rr := RDM(rr);
(* generate random date and randon dt *)
xdt := DWORD_TO_DT(rx);

(* analyze date *)
s1 := DT_TO_STRING(xdt);
s1 := RIGHT(s1, LEN(s1)-FIND(s1,'#'));
yr := STRING_TO_INT(LEFT(s1,4));
s1 := RIGHT(s1, LEN(s1)-FIND(s1,'-'));
mth := STRING_TO_INT(LEFT(s1,2));
s1 := RIGHT(s1, LEN(s1)-FIND(s1,'-'));
day := STRING_TO_INT(LEFT(s1,2));
(* analyze Time *)
s1 := RIGHT(s1, LEN(s1)-FIND(s1,'-'));
hr := STRING_TO_INT(LEFT(s1,2));
s1 := RIGHT(s1, LEN(s1)-FIND(s1,':'));
m := STRING_TO_INT(LEFT(s1,2));
s1 := RIGHT(s1, LEN(s1)-FIND(s1,':'));
sec := STRING_TO_INT(LEFT(s1,2));

(*
xd := DT_TO_DATE(xdt);
dt_to Date delivers wrong result when year > 2038
*)
xd := set_Date(yr,mth,day);

(* test set_date *)
test := 'set_date';
IF set_Date(yr,mth,day) <> xd THEN RETURN; END_IF;

(* test set_dt *)
test := 'set_dt';
IF set_DT(yr,mth,day,hr,m,sec) <> xdt THEN RETURN; END_IF;

(* test date_add *)
test := 'date_add';
YD := date_add(xd,0,0,0,0);
IF YD <> XD THEN RETURN; END_IF;
yd := date_add(d#2000-1-1,5,0,0,0);
IF yd <> d#2000-1-6 THEN RETURN; END_IF;
yd := date_add(d#2000-1-1,-31,0,0,0);
IF yd <> d#1999-12-1 THEN RETURN; END_IF;
yd := date_add(d#2000-1-1,60,0,0,0);
IF yd <> d#2000-3-1 THEN RETURN; END_IF;
yd := date_add(d#2001-1-1,59,0,0,0);
IF yd <> d#2001-3-1 THEN RETURN; END_IF;
yd := date_add(d#2002-1-1,59,0,0,0);
IF yd <> d#2002-3-1 THEN RETURN; END_IF;
yd := date_add(d#2003-1-1,59,0,0,0);
IF yd <> d#2003-3-1 THEN RETURN; END_IF;
yd := date_add(d#2004-1-1,60,0,0,0);
IF yd <> d#2004-3-1 THEN RETURN; END_IF;
yd := date_add(d#2000-1-1,0,1,0,0);
IF yd <> d#2000-1-8 THEN RETURN; END_IF;
yd := date_add(d#2000-1-1,0,-1,0,0);
IF yd <> d#1999-12-25 THEN RETURN; END_IF;
yd := date_add(d#2000-1-1,0,0,12,0);
IF yd <> d#2001-1-1 THEN RETURN; END_IF;
yd := date_add(d#2000-1-1,0,0,-1,0);
IF yd <> d#1999-12-1 THEN RETURN; END_IF;
yd := date_add(d#2000-1-1,0,0,0,99);
IF yd <> d#2099-1-1 THEN RETURN; END_IF;
yd := date_add(d#2000-1-1,0,0,0,-12);
IF yd <> d#1988-1-1 THEN RETURN; END_IF;
yd := date_add(d#2000-1-1,-31,1,1,1);
IF yd <> d#2001-1-8 THEN RETURN; END_IF;
yd := date_add(d#2000-1-1,31,1,-1,-1);
IF yd <> d#1999-1-8 THEN RETURN; END_IF;

(* test day_of_date *)
test := 'day_of_date';
IF day_of_date(XD) <> DATE_TO_DWORD(xd) / 86400 THEN RETURN; END_IF;

(* test day_of_month *)
test := 'day_of_month';
IF day_of_month(xd) <> day THEN RETURN; END_IF;

(* test day_of_year *)
test := 'day_of_year';
IF day_of_date(xd) - day_of_date(set_Date(yr,1,1)) + 1 <> day_of_year(xd) THEN RETURN; END_IF;

(* test days_delta *)
test := 'days_delta';
IF days_delta(xd, xd) <> 0 THEN RETURN; END_IF;
IF days_delta(D#2008-1-1,D#2007-12-31) <> -1 THEN RETURN; END_IF;
IF days_delta(D#2008-2-28,D#2008-3-1) <> 2 THEN RETURN; END_IF;
IF days_delta(D#2012-3-1,D#2012-2-28) <> -2 THEN RETURN; END_IF;
IF days_delta(D#2007-2-28,D#2007-3-1) <> 1 THEN RETURN; END_IF;
IF days_delta(D#1970-1-1,xd) <> day_of_date(xd) THEN RETURN; END_IF;

(* test DST *)
(*
Equation used TO calculate the beginning OF European Summer TIME:
Sunday (31 - (5*y/4 + 4) mod 7) March at 01.00 UTC
(valid through 2099, courtesy of Robert H. van Gent, EC).
European Summer Time ends (clocks go back) at 01.00 UTC on

    * 29 October 2006
    * 28 October 2007
    * 26 October 2008

Equation used to calculate the end of European Summer Time:
Sunday (31 - (5*y/4 + 1) mod 7) October at 01.00 UTC
(validity AND credits as above).
*)
test := 'dst';
ti := 31 -(5*yr/4 + 4) MOD 7;
te := 31-(5*yr/4+1) MOD 7;
tdt := set_DT(yr,3,ti,1,0,0);
tde := set_DT(yr,10,te,1,0,0);
tb := xdt >= tdt AND xdt < tde;
IF DST(xdt) <> tb THEN RETURN; END_IF;
IF DST(tdt) = FALSE THEN RETURN; END_IF;
tdt := set_DT(yr,3,ti,0,59,59);
IF DST(tdt) = TRUE THEN RETURN; END_IF;
tdt := set_DT(yr,10,te,0,59,59);
IF DST(tdt) = FALSE THEN RETURN; END_IF;
IF DST(tde) = TRUE THEN RETURN; END_IF;

(* easter test *)
test := 'easter';
IF easter_test() <> TRUE THEN RETURN; END_IF;

(* test leap_of_date *)
test := 'leap_of_Date';
tb := yr MOD 4 = 0;
IF leap_of_Date(xd) <> tb THEN RETURN; END_IF;

(* test leap_year *)
test := 'leap_year';
IF leap_year(yr) <> tb THEN RETURN; END_IF;

(* test local_time *)
test := 'local_time';
TT := T#12h;
IF local_time(xdt,-12,FALSE) <> xdt - TT THEN RETURN; END_IF;
IF local_time(xdt,0,FALSE) <> xdt THEN RETURN; END_IF;
TT := T#1h;
IF local_time(xdt,1,FALSE) <> xdt + TT THEN RETURN; END_IF;
TT := T#12h;
IF local_time(xdt,+12,FALSE) <> xdt + TT THEN RETURN; END_IF;
IF DST(xdt) THEN
	TT := T#11h;
	IF local_time(xdt,-12,TRUE) <> xdt - TT THEN RETURN; END_IF;
	TT := T#1h;
	IF local_time(xdt,0,TRUE) <> xdt + TT THEN RETURN; END_IF;
	TT := T#2h;
	IF local_time(xdt,1,TRUE) <> xdt + TT THEN RETURN; END_IF;
	TT := T#13h;
	IF local_time(xdt,+12,TRUE) <> xdt + TT THEN RETURN; END_IF;
ELSE
	TT := T#12h;
	IF local_time(xdt,-12,TRUE) <> xdt - TT THEN RETURN; END_IF;
	IF local_time(xdt,0,TRUE) <> xdt THEN RETURN; END_IF;
	TT := T#1h;
	IF local_time(xdt,1,TRUE) <> xdt + TT THEN RETURN; END_IF;
	TT := T#12h;
	IF local_time(xdt,+12,TRUE) <> xdt + TT THEN RETURN; END_IF;
END_IF;

(* ltime_to_utc *)
test := 'ltime_to_utc';
TT := T#1h;
IF Ltime_to_UTC(xdt+TT,FALSE,1) <> xdt THEN RETURN; END_IF;
IF Ltime_to_UTC(xdt - TT, FALSE,-1) <> xdt THEN RETURN; END_IF;
IF Ltime_to_UTC(xdt, FALSE,0) <> xdt THEN RETURN; END_IF;
TT := T#2h;
IF Ltime_to_UTC(xdt+ TT,TRUE,1) <> xdt THEN RETURN; END_IF;
IF Ltime_to_UTC(xdt, TRUE,-1) <> xdt THEN RETURN; END_IF;
TT := T#1h;
IF Ltime_to_UTC(xdt + TT, TRUE,0) <> xdt THEN RETURN; END_IF;

(* month test *)
test := 'month';
IF month(xd) <> mth THEN RETURN; END_IF;

(* period test *)
test := 'period';
yd := set_Date(2000,mth,day);
IF period(d#2000-3-3,xd,d#2000-9-3) <> (yd >= d#2000-3-3 AND yd <= d#2000-9-3) THEN RETURN; END_IF;
IF period(d#2000-9-3,xd,d#2000-3-3) <> (yd <= d#2000-3-3 OR yd >= d#2000-9-3) THEN RETURN; END_IF;

(* test weekday *)
test := 'weekday';
wd := weekday(xd);
wdi := DWORD_TO_DINT(DATE_TO_DWORD(xd)/86400);
wdi := (wdi + 4) MOD 7;
IF wdi = 0 THEN wdi := 7; END_IF;
IF wd <> wdi THEN RETURN; END_IF;

(* test year *)
test := 'year';
IF year(xd) <> yr THEN RETURN; END_IF;

(* test year_begin *)
test := 'year_begin';
IF year_begin(yr) <> set_Date(yr,1,1) THEN RETURN; END_IF;

(* test work_week *)
test := 'work_week';
IF NOT work_week_test() THEN RETURN; END_IF;

(* set output true if there are no errors *)
test := 'finished';
good := TRUE;


(* revision history
hm		26. mar. 2008		rev 1.0
	original release

*)
END_FUNCTION_BLOCK

(* POU Mathematical/RDMDW, ST *)
FUNCTION RDMDW : DWORD
VAR_INPUT
	last : DWORD;
END_VAR
VAR
	RX: REAL;
	M: REAL;
END_VAR




(*
version 1.0	14. mar 2008
programmer 	hugo
tested by		tobias

this function calculates a DWORD pseudo random number.

*)
M := BIT_COUNT(last);
RX := RDM(FRACT(M*pi1));
RDMDW := SHL(REAL_TO_DWORD(rx*65535),16);
RX := RDM(FRACT(M*e));
RDMDW := RDMDW OR (REAL_TO_DWORD(rx*65535) AND 16#0000FFFF);



(* revision history
hm		14. mar 2008		rev 1.0
	original version

*)
END_FUNCTION

(* POU Time&Date/set_Date, ST *)
FUNCTION set_Date : DATE
VAR_INPUT
	year : INT;
	month : INT;
	day : INT;
END_VAR
VAR
	count : DWORD;
END_VAR

(*
version 1.5	16. mar. 2008
programmer 	hugo
tested by		tobias

creates a date output from year, month and day of month   

*)
IF STEP7 THEN
	count := SHR(INT_TO_DWORD(year) * 1461 - 2907393,2)+INT_TO_DWORD(day);
ELSE
	count := SHR(INT_TO_DWORD(year) * 1461 - 2878173,2)+INT_TO_DWORD(day);
END_IF;

IF month < 5 THEN
	IF month < 3 THEN
		IF month = 2 THEN count := count + 31; END_IF;
	ELSE
		IF month = 4 THEN
			IF SHL(year,14) = 0 THEN count := count + 91; ELSE count := count + 90; END_IF;
		ELSE (* month = 3 *)
			IF SHL(year,14) = 0 THEN count := count + 60; ELSE count := count + 59; END_IF;
		END_IF;
	END_IF;
ELSIF month < 9 THEN
	IF month < 7 THEN
		IF month = 6 THEN
			IF SHL(year,14) = 0 THEN count := count + 152; ELSE count := count + 151; END_IF;
		ELSE (* month = 5 *)
			IF SHL(year,14) = 0 THEN count := count + 121; ELSE count := count + 120; END_IF;
		END_IF;
	ELSE
		IF month = 8 THEN
			IF SHL(year,14) = 0 THEN count := count + 213; ELSE count := count + 212; END_IF;
		ELSE (* month = 7 *)
			IF SHL(year,14) = 0 THEN count := count + 182; ELSE count := count + 181; END_IF;
		END_IF;
	END_IF;
ELSE (* month is 9 or higher *)
	IF month < 11 THEN
		IF month = 10 THEN
			IF SHL(year,14) = 0 THEN count := count + 274; ELSE count := count + 273; END_IF;
		ELSE (* month = 9 *)
			IF SHL(year,14) = 0 THEN count := count + 244; ELSE count := count + 243; END_IF;
		END_IF;
	ELSE
		IF month = 12 THEN
			IF SHL(year,14) = 0 THEN count := count + 335; ELSE count := count + 334; END_IF;
		ELSE (* month = 11 *)
			IF SHL(year,14) = 0 THEN count := count + 305; ELSE count := count + 304; END_IF;
		END_IF;
	END_IF;
END_IF;
set_Date := DWORD_TO_DATE(count * 86400);

(*  code before rev 1.4
leap := leap_year(year);
IF STEP7 THEN
	count := SHR((year-1)*1461-2905932+day*4,2);
ELSE
	count := SHR((year-1)*1461-2876712+day*4,2);
END_IF;
CASE month OF
2:	count := count + 31;
3:	IF leap THEN count := count + 60; ELSE count := count + 59; END_IF;
4:	IF leap THEN count := count + 91; ELSE count := count + 90; END_IF;
5:	IF leap THEN count := count + 121; ELSE count := count + 120; END_IF;
6:	IF leap THEN count := count + 152; ELSE count := count + 151; END_IF;
7:	IF leap THEN count := count + 182; ELSE count := count + 181; END_IF;
8:	IF leap THEN count := count + 213; ELSE count := count + 212; END_IF;
9:	IF leap THEN count := count + 244; ELSE count := count + 243; END_IF;
10:	IF leap THEN count := count + 274; ELSE count := count + 273; END_IF;
11:	IF leap THEN count := count + 305; ELSE count := count + 304; END_IF;
12:	IF leap THEN count := count + 335; ELSE count := count + 334; END_IF;
END_CASE;
set_Date := DWORD_TO_DATE(count * 86400);
*)

(* old code before rev 1.3
leap := leap_year(year);
IF STEP7 THEN
	count := TRUNC((year-1)*365.25-726483+day);
ELSE
	count := TRUNC((year-1)*365.25-719178+day);
END_IF;
CASE month OF
2:	count := count + 31;
3:	IF leap THEN count := count + 60; ELSE count := count + 59; END_IF;
4:	IF leap THEN count := count + 91; ELSE count := count + 90; END_IF;
5:	IF leap THEN count := count + 121; ELSE count := count + 120; END_IF;
6:	IF leap THEN count := count + 152; ELSE count := count + 151; END_IF;
7:	IF leap THEN count := count + 182; ELSE count := count + 181; END_IF;
8:	IF leap THEN count := count + 213; ELSE count := count + 212; END_IF;
9:	IF leap THEN count := count + 244; ELSE count := count + 243; END_IF;
10:	IF leap THEN count := count + 274; ELSE count := count + 273; END_IF;
11:	IF leap THEN count := count + 305; ELSE count := count + 304; END_IF;
12:	IF leap THEN count := count + 335; ELSE count := count + 334; END_IF;
END_CASE;
set_Date := DWORD_TO_DATE(count * 86400);
*)




(* revision history
hm	4. aug. 2006	rev 1.0
	original version

hm	19 sep. 2007	rev 1.1
	use function leap_year to calculate leap year, more exceptions are handled

hm	1. okt	2007	rev 1.2
	added compatibility to step7

hm	16.dec 2007	rev 1.3
	changed code to improove performance

hm	3. jan. 2008	rev 1.4
	further improvements in performance

hm	16. mar. 2008	rev 1.5
	added type conversions to avoid warnings under codesys 3.0
*)
END_FUNCTION

(* POU Time&Date/year, ST *)
FUNCTION year : INT
VAR_INPUT
	idate : DATE;
END_VAR
VAR
END_VAR

(*
version 1.2	23 dec 2007
programmer 	hugo
tested by		tobias

returs the year of a date  
the function works for dates from 1970 - 2099 

*)
IF Step7 THEN
	year := DWORD_TO_INT((DATE_TO_DWORD(idate)+43200) / 31557600 + 1990);
ELSE
	year := DWORD_TO_INT((DATE_TO_DWORD(idate)+43200) / 31557600 + 1970);
END_IF;

(* code used prior to rev 1.1
year := DWORD_TO_INT((DATE_TO_DWORD(idate)/864+71954300)/36525);
*)

(* revision history
hm	4. aug 2006		rev 1.0
	original version

hm	1. okt 2007		rev 1.1
	corrected error in algorithm
	adjustment for S7 compatibility

hm	23.12.2007		rev 1.2
	changed code for better performance
*)
END_FUNCTION

(* POU Time&Date/month, ST *)
FUNCTION month : INT
VAR_INPUT
	idate : DATE;
END_VAR
VAR
END_VAR

(*
version 1.1	1 okt 2007
programmer 	hugo
tested by		tobias

returns the month of a year

*)
month := day_of_year(idate);
IF leap_of_Date(idate) THEN
	CASE month OF
		1..31 	:	month := 1;
		32..60	:	month := 2;
		61..91	:	month := 3;
		92..121 :	month := 4;
		122..152:	month := 5;
		153..182:	month := 6;
		183..213:	month := 7;
		214..244:	month := 8;
		245..274:	month := 9;
		275..305:	month := 10;
		306..335:	month := 11;
		336..366:	month := 12;
	END_CASE;
ELSE
	CASE month OF
		1..31 	:	month := 1;
		32..59	:	month := 2;
		60..90	:	month := 3;
		91..120 :	month := 4;
		121..151:	month := 5;
		152..181:	month := 6;
		182..212:	month := 7;
		213..243:	month := 8;
		244..273:	month := 9;
		274..304:	month := 10;
		305..334:	month := 11;
		335..365:	month := 12;
	END_CASE;
END_IF;


(* old code used in rev 1.0
month := STRING_TO_INT(MID(DATE_TO_STRING(idate),2,8));
*)

(* revision history
hm	1. aug 2006		rev 1.0
	original version	

hm	1. okt 2007		rev 1.1
	replaced old code (string conversion) with mathematics
	the execution time is now multiple times faster.

*)
END_FUNCTION

(* POU Time&Date/day_of_year, ST *)
FUNCTION day_of_year : INT
VAR_INPUT
	idate : DATE;
END_VAR
VAR
END_VAR

(*
version 1.2	4 jan 2008
programmer 	hugo
tested by		tobias

calculates the day of the year

*)
day_of_year := DWORD_TO_INT((DATE_TO_DWORD(idate) - DATE_TO_DWORD(year_begin(year(idate))))/86400) + 1;


(* version before rev 1.2
IF step7 THEN
	day_of_year := DWORD_TO_INT(DATE_TO_DWORD(idate)/86400 + 726483 - TRUNC((year(idate)-1)*365.25));
ELSE
	day_of_year := DWORD_TO_INT(DATE_TO_DWORD(idate)/86400 + 719178 - TRUNC((year(idate)-1)*365.25));
END_IF;
*)


(* revivision history
hm	4. aug 2007		rev 1.0
	original version

hm	1. okt 2007		rev 1.1
	added compatibility to STEP7

hm	4. jan 2008		rev 1.2
	changed code for better performance
*)
END_FUNCTION

(* POU Time&Date/year_begin, ST *)
FUNCTION year_begin : DATE
VAR_INPUT
	y : INT;
END_VAR
VAR
END_VAR

(*
version 1.1	4. Jan 2008
programmer 	hugo
tested by		tobias

returs the date of january 1st for the given year  
the function works for dates from 1970 - 2099 

*)
IF Step7 THEN
	year_begin := DWORD_TO_DATE(SHR(INT_TO_DWORD(y) * 1461 - 2907389,2)*86400);
ELSE
	year_begin := DWORD_TO_DATE(SHR(INT_TO_DWORD(y) * 1461 - 2878169,2)*86400);
END_IF;

(* revision history
hm	19. dec 2007	rev 1.0
	original version

hm	4. jan 2008	rev 1.1
	formula for step7 was incorrect during leap years

*)
END_FUNCTION

(* POU Time&Date/leap_of_Date, ST *)
FUNCTION leap_of_Date : BOOL
VAR_INPUT
	idate : DATE;
END_VAR
VAR
END_VAR

(*
version 1.2	8 jan 2008
programmer 	hugo
tested by		tobias

leap_year is true if the tested year is a leap year  

*)
leap_of_Date := SHL(DWORD_TO_INT((DATE_TO_DWORD(idate)+43200) / 31557600)+2,14) = 0;


(* change history

2.10.2006		rev 1.1
the function now calls leap_year to accomodate further accuracy.
the function now works for any year from 1970 to 2100

8. jan 2008		rev 1.2
	improved code for better performance
*)
END_FUNCTION

(* POU Time&Date/set_DT, ST *)
FUNCTION set_DT : DT
VAR_INPUT
	year : INT;
	month : INT;
	day : INT;
	hour : INT;
	minute : INT;
	second : INT;
END_VAR
VAR
END_VAR

(*
version 1.5	16 mar 2008
programmer 	hugo
tested by		tobias


creates a date output from year, month and day of month
year must be in the form of 4 digits ie 2006 or 1977.
*)
set_DT := DWORD_TO_DT(DATE_TO_DWORD(set_Date(year, month, day)) + INT_TO_DWORD(second) + INT_TO_DWORD(minute) * 60 + INT_TO_DWORD(hour) * 3600);


(* revision history
hm	4. aug. 2006		rev 1.0
	original version

hm		19 sep. 2007	rev 1.1
	use function leap_year to calculate leap year, more exceptions are handled

hm		1. okt 2007		rev 1.2
	added step7 compatibility
	call function set_date

hm		8. oct 2007		rev 1.3
	deleted unused variables count and leap

hm		1. 11 2007		rev 1.4
	converted hour type integer to dword in calculation to avoid overrun on möller ecp4

hm		16. mar 2008	rev 1.5
	added type conversions to avoid warnings under codesys 3.0
*)
END_FUNCTION

(* POU Time&Date/hour, ST *)
FUNCTION hour : INT
VAR_INPUT
	itod : TOD;
END_VAR
VAR
END_VAR

(*
version 1.1	2 okt 2006
programmer 	hugo
tested by		tobias

extracts the hour of a Time_of_day 
*)
hour := DWORD_TO_INT(TOD_TO_DWORD(itod)/3600000);


(* change history
hm 4. aug 2006	rev 1.0
	original version

hm 2.10.2006 	rev 1.1
	changed name of input to itod

*)
END_FUNCTION

(* POU Time&Date/minute, ST *)
FUNCTION minute : INT
VAR_INPUT
	itod : TOD;
END_VAR
VAR
END_VAR

(*
version 1.1	2 oct 2006
programmer 	hugo
tested by		tobias

extracts the minutes out of TOD truncating the ceconds 

*)  
minute := DWORD_TO_INT(TOD_TO_DWORD(itod)/60000 - TOD_TO_DWORD(itod)/3600000 * 60);


(* change history

2.10.2006 changes name of input to itod

*)
END_FUNCTION

(* POU Time&Date/second, ST *)
FUNCTION second : REAL
VAR_INPUT
	itod : TOD;
END_VAR
VAR
END_VAR

(*
version 1.1	2 oct 2006
programmer 	hugo
tested by		tobias

returns the seconds and milliseconds as real of TOD   
execution time on wago 750-841 = 20 us 
*)
second := DWORD_TO_REAL(TOD_TO_DWORD(itod) - TOD_TO_DWORD(itod)/60000 * 60000)/1000;



(* change history

2.10.2006 changes name of input to itod

*)
END_FUNCTION

(* POU Time&Date/date_add, ST *)
FUNCTION date_add : DATE
VAR_INPUT
	idate : DATE;
	D : INT;
	W : INT;
	M : INT;
	Y : INT;
END_VAR
VAR
	mo: INT;
	yr : INT;
END_VAR


(*
version 1.3	22. mar 2008
programmer 	hugo
tested by		tobias

date_add adds days, weeks, month or years to a date.
negative inputs are allowed for subtraction.

*)
date_add := DWORD_TO_DATE(DATE_TO_DWORD(idate) + 86400 * INT_TO_DWORD(d) + 604800 * INT_TO_DWORD(w));
mo := month(date_add);
yr := year(date_add) + y + FLOOR(INT_TO_REAL(mo + m - 1) / 12.0);
mo := mo + (ABS(m) MOD 12) * SGN(m);
IF mo < 1 THEN
	mo := mo + 12;
ELSIF mo > 12 THEN
	mo := mo - 12;
END_IF;
date_add := set_Date(yr,mo,day_of_month(date_add));



(* revision history

hm 27.12.2006		rev 1.0

hm 12.4.2007		rev 1.1
	corrected an error while date would be incorrect when year  = 0

hm	1.11.2007		rev 1.2
	added int_to_dword stetements to avoid possible overrun with möller ecp4

hm	22. mar. 2008	rev 1.3
	fixed some bugs when month was negative
*)
END_FUNCTION

(* POU Mathematical/SGN, ST *)
FUNCTION SGN : INT
VAR_INPUT
	X : REAL;
END_VAR
VAR
END_VAR

(*
version 1.1	11 nov 2007
programmer 	hugo
tested by	tobias

sgn returns 0 when X = 0 , -1 when X < 1 and +1 when X > 1

*)
IF X > 0 THEN
	sgn := 1;
ELSIF X < 0 THEN
	sgn := -1;
ELSE
	sgn := 0;
END_IF;

(* revision histroy
hm	16. oct 2007	rev 1.0
	original version

hm	11. nov 2007	rev 1.1
	changed type of function from real to int
*)
END_FUNCTION

(* POU Time&Date/day_of_month, ST *)
FUNCTION day_of_month : INT
VAR_INPUT
	idate : DATE;
END_VAR
VAR
END_VAR

(*
version 1.4	8. jan 2008
programmer 	hugo
tested by		tobias

returns the day OF month for any DATE

*)
day_of_month := day_of_year(idate);
IF leap_of_Date(idate) THEN
	CASE day_of_month OF
		32..60	:	day_of_month := day_of_month - 31;
		61..91	:	day_of_month := day_of_month - 60;
		92..121 :	day_of_month := day_of_month - 91;
		122..152:	day_of_month := day_of_month - 121;
		153..182:	day_of_month := day_of_month - 152;
		183..213:	day_of_month := day_of_month - 182;
		214..244:	day_of_month := day_of_month - 213;
		245..274:	day_of_month := day_of_month - 244;
		275..305:	day_of_month := day_of_month - 274;
		306..335:	day_of_month := day_of_month - 305;
		336..366:	day_of_month := day_of_month - 335;
	END_CASE;
ELSE
	CASE day_of_month OF
		32..59	:	day_of_month := day_of_month - 31;
		60..90	:	day_of_month := day_of_month - 59;
		91..120 :	day_of_month := day_of_month - 90;
		121..151:	day_of_month := day_of_month - 120;
		152..181:	day_of_month := day_of_month - 151;
		182..212:	day_of_month := day_of_month - 181;
		213..243:	day_of_month := day_of_month - 212;
		244..273:	day_of_month := day_of_month - 243;
		274..304:	day_of_month := day_of_month - 273;
		305..334:	day_of_month := day_of_month - 304;
		335..365:	day_of_month := day_of_month - 334;
	END_CASE;
END_IF;


(*
this function is simple but took too long with 133 us
the problem is date_to_string is far too slow
day_of_month := STRING_TO_INT(RIGHT(DATE_TO_STRING(idate),2));

Revision history

hm 22.1.2007		rev 1.1
	deleted unused variable day_in_year and day_in_year_begin

hm	1. okt 2007		rev 1.2
	changed code to use day_of_year and leap_of_date
	added compatibility to STEP7

hm	8. oct 2007		rev 1.3
	deleted unused variable yr

hm	8. jan 2008		rev 1.4
	improved performance
*)
END_FUNCTION

(* POU Time&Date/day_of_date, ST *)
FUNCTION day_of_date : DINT
VAR_INPUT
	idate : DATE;
END_VAR
VAR
END_VAR


(*
	version 1.2	22. mar. 2008
	programmer 	oscat
	tested BY		oscat

DAY_OF_DATE returns the days since 1.1.1970

*)
IF STEP7 THEN
	(* adjust step7 day by 7305 days because step7 date fornat starts at 1.1.1990  *)
	day_of_date := DWORD_TO_DINT(DATE_TO_DWORD(idate) / 86400) + 7305;
ELSE
	day_of_date := DWORD_TO_DINT(DATE_TO_DWORD(idate) / 86400);
END_IF;


(* revision history
hm		16.9.2007		rev 1.0
	original version

hm		1. okt 2007		rev 1.1
	added step7 compatibility

hm		22. mar. 2008	rev 1.2
	changed output from int to Dint because the total date range is 49710 days

*)
END_FUNCTION

(* POU Time&Date/days_delta, ST *)
FUNCTION days_delta : DINT
VAR_INPUT
	date_1 : DATE;
	date_2 : DATE;
END_VAR
VAR
END_VAR

(*
version 1.2	22. mar. 2008
programmer 	hugo
tested by		tobias

days_delta calculates the days between two dates. the days are calculated date_2 - date_1.

*)
days_delta := day_of_date(date_2) - day_of_date(date_1);

(* revision history
hm	27. dec 2006	rev 1.0
	original version

hm	16.9.2007		rev 1.1
	coorected an error in formula and changed algorithm to show positive and negative delta

hm	22. mar. 2008	rev 1.2
	changed output from int to dint because the total date range is 49710 days
*)
END_FUNCTION

(* POU Time&Date/DST, ST *)
FUNCTION DST : BOOL
VAR_INPUT
	utc : DT;
END_VAR
VAR
	yr : INT;
	yr4 : DWORD;
	ltc: DWORD;
	idate : DWORD;
END_VAR

(*
version 1.3	16. mar. 2008
programmer 	hugo
tested by		tobias

this functions returns TRUE IF dst TIME is active 
the FUNCTION calculates automatically for any year betweek 1970 AND 2099 
wheather daylight savings is on OR off 
the summertime calculation is done according to european standards.
dst will become TRUE AT 01:00 utc in the morning FOR the respective days 
AND it will become FALSE after daylight savings TIME is switched back end OF october at 01:00 utc

*)
yr := year(DT_TO_DATE(utc));
ltc := DT_TO_DWORD(utc);
idate := DT_TO_DWORD(set_DT(yr,3,31,1,0,0));
yr4 := SHR(5*INT_TO_DWORD(yr),2);
DST := (idate - ((yr4+4) MOD 7)*86400 <= ltc) AND (idate + (214 - (yr4+1) MOD 7)*86400 > ltc);

(* revision history
hm	4. aug 2006	rev 1.0
	original version

hm	24. okt 2007	rev 1.1
	deleted time_zone_offset input because dst is generally at 01:00 utc and not mesz
	uk starts 01:00 utc and also greece

hm	1. dec 2007	rev 1.2
	changed code to improve performance

hm	16. mar. 2008	rev 1.3
	added type conversion to avoid warnings under codesys 3.0
	code improvement for better performance

*)

(*
Equation used TO calculate the beginning OF European Summer TIME:
Sunday (31 - (5*y/4 + 4) mod 7) March at 01.00 UTC
(valid through 2099, courtesy of Robert H. van Gent, EC).

European Summer Time ends (clocks go back) at 01.00 UTC on

    * 29 October 2006
    * 28 October 2007
    * 26 October 2008

Equation used to calculate the end of European Summer Time:
Sunday (31 - (5*y/4 + 1) mod 7) October at 01.00 UTC
(validity AND credits as above).

*)
END_FUNCTION

(* POU XTEST/Testprojekt/TEST Routines/easter_test, ST *)
FUNCTION easter_test : BOOL
VAR_INPUT
END_VAR
VAR
	x: BOOL := TRUE;
END_VAR
x := easter(1980) = d#1980-4-6;
x := easter(1981) = d#1981-4-19 AND x;
x := easter(1982) = d#1982-4-11 AND x;
x := easter(1983) = d#1983-4-3 AND x;
x := easter(1984) = d#1984-4-22 AND x;
x := easter(1985) = d#1985-4-7 AND x;
x := easter(1986) = d#1986-3-30 AND x;
x := easter(1987) = d#1987-4-19 AND x;
x := easter(1988) = d#1988-4-3 AND x;
x := easter(1989) = d#1989-3-26 AND x;
x := easter(1990) = d#1990-4-15 AND x;
x := easter(1991) = d#1991-3-31 AND x;
x := easter(1992) = d#1992-4-19 AND x;
x := easter(1993) = d#1993-4-11 AND x;
x := easter(1994) = d#1994-4-3 AND x;
x := easter(1995) = d#1995-4-16 AND x;
x := easter(1996) = d#1996-4-7 AND x;
x := easter(1997) = d#1997-3-30 AND x;
x := easter(1998) = d#1998-4-12 AND x;
x := easter(1999) = d#1999-4-4 AND x;
x := easter(2000) = d#2000-4-23 AND x;
x := easter(2001) = d#2001-4-15 AND x;
x := easter(2002) = d#2002-3-31 AND x;
x := easter(2003) = d#2003-4-20 AND x;
x := easter(2004) = d#2004-4-11 AND x;
x := easter(2005) = d#2005-3-27 AND x;
x := easter(2006) = d#2006-4-16 AND x;
x := easter(2007) = d#2007-4-8 AND x;
x := easter(2008) = d#2008-3-23 AND x;
x := easter(2009) = d#2009-4-12 AND x;
x := easter(2010) = d#2010-4-4 AND x;
x := easter(2011) = d#2011-4-24 AND x;
x := easter(2012) = d#2012-4-8 AND x;
x := easter(2013) = d#2013-3-31 AND x;
x := easter(2014) = d#2014-4-20 AND x;
x := easter(2015) = d#2015-4-5 AND x;
x := easter(2016) = d#2016-3-27 AND x;
x := easter(2017) = d#2017-4-16 AND x;
x := easter(2018) = d#2018-4-1 AND x;
x := easter(2019) = d#2019-4-21 AND x;
x := easter(2020) = d#2020-4-12 AND x;
x := easter(2021) = d#2021-4-4 AND x;
x := easter(2022) = d#2022-4-17 AND x;
x := easter(2023) = d#2023-4-9 AND x;
x := easter(2024) = d#2024-3-31 AND x;
x := easter(2025) = d#2025-4-20 AND x;
x := easter(2026) = d#2026-4-5 AND x;
x := easter(2027) = d#2027-3-28 AND x;
x := easter(2028) = d#2028-4-16 AND x;
x := easter(2029) = d#2029-4-1 AND x;
x := easter(2030) = d#2030-4-21 AND x;
x := easter(2031) = d#2031-4-13 AND x;
x := easter(2032) = d#2032-3-28 AND x;
x := easter(2033) = d#2033-4-17 AND x;
x := easter(2034) = d#2034-4-9 AND x;
x := easter(2035) = d#2035-3-25 AND x;
x := easter(2036) = d#2036-4-13 AND x;
x := easter(2037) = d#2037-4-5 AND x;
x := easter(2038) = d#2038-4-25 AND x;
x := easter(2039) = d#2039-4-10 AND x;
x := easter(2040) = d#2040-4-1 AND x;
x := easter(2041) = d#2041-4-21 AND x;
x := easter(2042) = d#2042-4-6 AND x;
x := easter(2043) = d#2043-3-29 AND x;
x := easter(2044) = d#2044-4-17 AND x;
x := easter(2045) = d#2045-4-9 AND x;
x := easter(2046) = d#2046-3-25 AND x;
x := easter(2047) = d#2047-4-14 AND x;
x := easter(2048) = d#2048-4-5 AND x;
x := easter(2049) = d#2049-4-18 AND x;
x := easter(2050) = d#2050-4-10 AND x;
x := easter(2051) = d#2051-4-2 AND x;
x := easter(2052) = d#2052-4-21 AND x;
x := easter(2053) = d#2053-4-6 AND x;
x := easter(2054) = d#2054-3-29 AND x;
x := easter(2055) = d#2055-4-18 AND x;
x := easter(2056) = d#2056-4-2 AND x;
x := easter(2057) = d#2057-4-22 AND x;
x := easter(2058) = d#2058-4-14 AND x;
x := easter(2059) = d#2059-3-30 AND x;
x := easter(2060) = d#2060-4-18 AND x;
x := easter(2061) = d#2061-4-10 AND x;
x := easter(2062) = d#2062-3-26 AND x;
x := easter(2063) = d#2063-4-15 AND x;
x := easter(2064) = d#2064-4-6 AND x;
x := easter(2065) = d#2065-3-29 AND x;
x := easter(2066) = d#2066-4-11 AND x;
x := easter(2067) = d#2067-4-3 AND x;
x := easter(2068) = d#2068-4-22 AND x;
x := easter(2069) = d#2069-4-14 AND x;
x := easter(2070) = d#2070-3-30 AND x;
x := easter(2071) = d#2071-4-19 AND x;
x := easter(2072) = d#2072-4-10 AND x;
x := easter(2073) = d#2073-3-26 AND x;
x := easter(2074) = d#2074-4-15 AND x;
x := easter(2075) = d#2075-4-7 AND x;
x := easter(2076) = d#2076-4-19 AND x;
x := easter(2077) = d#2077-4-11 AND x;
x := easter(2078) = d#2078-4-3 AND x;
x := easter(2079) = d#2079-4-23 AND x;
x := easter(2080) = d#2080-4-7 AND x;
x := easter(2081) = d#2081-3-30 AND x;
x := easter(2082) = d#2082-4-19 AND x;
x := easter(2083) = d#2083-4-4 AND x;
x := easter(2084) = d#2084-3-26 AND x;
x := easter(2085) = d#2085-4-15 AND x;
x := easter(2086) = d#2086-3-31 AND x;
x := easter(2087) = d#2087-4-20 AND x;
x := easter(2088) = d#2088-4-11 AND x;
x := easter(2089) = d#2089-4-3 AND x;
x := easter(2090) = d#2090-4-16 AND x;
x := easter(2091) = d#2091-4-8 AND x;
x := easter(2092) = d#2092-3-30 AND x;
x := easter(2093) = d#2093-4-12 AND x;
x := easter(2094) = d#2094-4-4 AND x;
x := easter(2095) = d#2095-4-24 AND x;
x := easter(2096) = d#2096-4-15 AND x;
x := easter(2097) = d#2097-3-31 AND x;
x := easter(2098) = d#2098-4-20 AND x;
x := easter(2099) = d#2099-4-12 AND x;
easter_test := X;

(* revision history
hm		26. mar. 2008		rev 1.0
	original release

*)
END_FUNCTION

(* POU Time&Date/easter, ST *)
FUNCTION easter : DATE
VAR_INPUT
	year : INT;
END_VAR
VAR
	b,c: INT;
	oday: INT;
	omon: INT;
END_VAR

(*
version 1.2	3. feb 2008
programmer 	hugo
tested by		tobias

easter calculates the day of easter sunday for a given year.
most other catholic holidays are calculated in reference to easter sunday.

*)
(* this algorithms is 60 us *)

b := (204 - 11 * (year MOD 19)) MOD 30;
IF b > 27 THEN b := b - 1; END_IF;
c := (year + SHR(year,2) + b - 13) MOD 7;
oday := 28 + b - c;
IF oday > 33 THEN
    oday := oday - 31;
    omon := 4;
ELSE
	omon := 3;
END_IF;
easter := set_Date(year, omon, oday);



(* alternativer algorithmus ueber das pasah fest
execution time roughly 200us
Der sog. Passah-Vollmond wird berechnet, in dem das Jahr durch 19 ge-
teilt wird und der Rest mit der folgenden Tabelle verglichen wird:
 
    0: Apr 14       5: Apr 18      10: Mrz 25      15: Mrz 30
    1: Apr 03       6: Apr 08      11: Apr 13      16: Apr 17
    2: Mrz 23       7: Mrz 28      12: Apr 02      17: Apr 07
    3: Apr 11       8: Apr 16      13: Mrz 22      18: Mrz 27
    4: Mrz 31       9: Apr 05      14: Apr 10
 
Faellt dieses Datum auf einen Sonntag, ist Ostern der naechste Sonntag!
 
Beispiel: 1992 MOD 19 = 16, daraus folgt 17.04., der naechste Sonntag
          ist dann der 19. April (Ostersonntag)
*)


(* this algorithm is 180 us
a := year MOD 19;
b := year / 100;
c := year MOD 100;
d := b / 4;
e := b MOD 4;
f := (b + 8) / 25;
g := (b - f + 1) / 3;
h := (19 * a + b - d -g + 15) MOD 30;
i := C / 4;
k := c MOD 4;
l := (32 + 2*e + 2*i - h - k) MOD 7;
m := (a + 11 * h + 22 * l) / 451;
x := h + l - 7 * m + 114;
n := X / 31;
o := x MOD 31 + 1;

easter := set_Date(year,n,o);
*)
(*
Im Magazin "Nature" vom 20. April 1876 veröffentlichte ein anonymer Autor eine Tabelle mit Regeln zur Berechnung des (Gregorianischen) Ostersonntages des Jahres J. In Formeln ausgedrückt erhält man das Folgende:
a	=	J mod 19
b	=	int(J / 100)
c	=	J mod 100
d	=	int(b / 4)
e	=	b mod 4
f	=	int((b + 8) / 25)
g	=	int((b - f + 1) / 3
h	=	(19 · a + b - d - g + 15) mod 30
i	=	int(c / 4)
k	=	c mod 4
l	=	(32 + 2 · e + 2 · i - h - k) mod 7
m	=	int((a + 11 · h + 22 · l) / 451)
n	=	int((h + l - 7 · m + 114) / 31)
o	=	(h + l - 7 · m + 114) mod 31

n ist hierbei die Nummer des Monats, o + 1 die Nummer des Tages auf welchen der Ostersonntag im Jahr J fällt. Dieser Algorithmus kommt ohne Hilfszahlen aus.

*)

(* revision history
hm	27. dec 2006	rev 1.0
	original version

hm	15. dec 2007	rev 1.1
	modified code for better performance

hm	3. feb 2008		rev 1.2
	modified code for better performance
*)
END_FUNCTION

(* POU Time&Date/leap_year, ST *)
FUNCTION leap_year : BOOL
VAR_INPUT
	yr : INT;
END_VAR
VAR
END_VAR

(*
version 1.1	2 oct 2006
programmer 	hugo
tested by		tobias


leap_year is true if the tested year is a leap year  
  
*)
leap_year := SHL(yr,14) = 0;

(* this code was used prior to rev 1.1

IF yr MOD 400 = 0 THEN leap_year := TRUE;
ELSIF yr MOD 100 = 0 THEN leap_year := FALSE;
ELSIF yr MOD 4 =0 THEN leap_year := TRUE;
ELSE leap_year := FALSE;
END_IF;

*)

(* change history

hm 	2.10.2006		rev 1.1
	the function now works for any year from 1970 up to 2100

hm	1. oct 2007		rev 1.2
	chaged code for higher performance
*)
END_FUNCTION

(* POU Time&Date/local_time, ST *)
FUNCTION local_time : DT
VAR_INPUT
	utc : DT;
	time_zone_offset : INT;
	dst_enable: BOOL;
END_VAR
VAR
	tx : TIME;
END_VAR

(*
version 1.4	8 dec 2007
programmer 	hugo
tested by		tobias

localtime calculates the local time according to DSTenable and time_zone_offset.
the dst input only tells the function the dst (daylight savings time) is enabled but the calculation for summertime on and off is done by the function itself.
this means the dst input only tells the function to switch summertime on and off automatically or not.
the function will switch to summertime automatically at the specified time end of march and back end of october.
the summertime calculation is done according to european standards.
the input is world time (UTC) and a given time_zone_offset for any time_zone.

*)
tx := DWORD_TO_TIME(INT_TO_DWORD(ABS(time_zone_offset))* 3600000);

IF DST(utc) AND dst_enable THEN
	IF time_zone_offset < 0 THEN local_time := utc - tx + T#1h; ELSE local_time := utc + tx + T#1h; END_IF;
ELSE
	IF time_zone_offset < 0 THEN local_time := utc - tx; ELSE local_time := utc + tx; END_IF;
END_IF;


(*

change history

2.10.2006 hm	rev 1.1
	corrected an error in the dst check for correct function

24. oct 2007	rev 1.2
	changed dst calculation because function dst was upgraded no error in DCF77 only a change in DST

12. nov 2007	rev 1.3
	changed time_zone_offset from time to integer to allow for negative offset time zones

8 dec 2007		rev 1.4
	corrected a problem with time_zone_offset
*)
END_FUNCTION

(* POU Time&Date/Ltime_to_UTC, ST *)
FUNCTION Ltime_to_UTC : DT
VAR_INPUT
	Ltime : DT;
	DST : BOOL;
	Time_Zone_Offset : INT;
END_VAR
VAR
	dst_offset : TIME := T#1h;
	tx: TIME;
END_VAR

(*
version 1.3		8 dec 2007
programmer 	hugo
tested by		tobias

LTIME_TO_UTC calculates UTC (World Time) from a local time LTIME. utc is calculated 
by subtracting Time_Zone_Offset from ltime and if dst it true subtracting an additional hour from ltime.

*)
(* convert integer time_zone_offset to hours *)
tx := DWORD_TO_TIME(INT_TO_DWORD(ABS(time_zone_offset))* 3600000);

IF DST THEN
	IF time_zone_offset < 0 THEN
		Ltime_to_UTC := Ltime + tx - dst_offset;
	ELSE
		Ltime_to_UTC := Ltime - tx - dst_offset;
	END_IF;
ELSE
	IF time_zone_offset < 0 THEN
		Ltime_to_UTC := Ltime + tx;
	ELSE
		Ltime_to_UTC := Ltime - tx;
	END_IF;
END_IF;



(* revision history
hm 5.7.2007		rev 1.0		
	original version

hm 5.11.2007	rev 1.1
	replaced literal constant with variable because of error in möller ecp4 compiler

hm	12.nov 2007	rev 1.2
	changed Type of time_zone_offset from time to int to allow for time zones with negative offset

hm	8. dec 2007	rev 1.3
	corrected a problem with time_zone_offset
*)
END_FUNCTION

(* POU Time&Date/Ltime, ST *)
FUNCTION_BLOCK Ltime
VAR_INPUT
	UTC : DT;
	dst_enable : BOOL;
	time_zone_offset : INT;
END_VAR
VAR_OUTPUT
	local_DT : DT;
	DST_on : BOOL;
	wday : INT;
END_VAR
VAR
	tx: TIME;
END_VAR

(*

version 1.6	8 dec 2007
programmer 	oscat
tested by		tobias

ltime is a real time clock that uses the system rtc as utc time and calculates and given time zone.
the utc time is supplied on the input UTC.
according to the input variable time_zone_offset when the input dst_enable is true,
the dst on and off times are calculated by a formula for any given year and the time is advanced and reset by one hour
at 02:00 and 03:00 for the last sunday of march and last sunday of october.
the code is high performance and the rtc counts every second.
if more then one time zone is needed by the systen the clock can be started many times by placing more then one function block.

execution time on wago 750-841 = 20 us 
 
*)
tx := DWORD_TO_TIME(INT_TO_DWORD(ABS(time_zone_offset))* 3600000);
DST_ON := DST(UTC) AND dst_enable;
IF DST_ON THEN
	IF time_zone_offset < 0 THEN local_DT := UTC - tx + t#1h; ELSE local_DT := UTC + tx + t#1h; END_IF;
ELSE
	IF time_zone_offset < 0 THEN local_DT := UTC - tx; ELSE local_DT := UTC + tx; END_IF;
END_IF;
wday := weekday(DT_TO_DATE(local_DT));


(* revision history

hm 2.10.2006	rev 1.1
	corrected an error where dst would be delayed by 0.1second

hm 17.1.2007	rev 1.2
	added utc input instead of internal sysrtcgettime because this would only work on wago.
	dst_enable would not be checked before dst would be enabled.

hm 18.3.2007	rev 1.3
	changed code, dst would not work during first cycle.

hm 24.10.2007	rev 1.4
	changed code because the execution every 100ms can cause major problems if the supplied time was not correct at start.
	use of new dst function

hm 12. nov 2007	rev 1.5
		changed Type of time_zone_offset from time to int to allow for time zones with negative offset

8 dec 2007		rev 1.6
	corrected a problem with time_zone_offset
*)
END_FUNCTION_BLOCK

(* POU Time&Date/weekday, ST *)
FUNCTION weekday : INT
VAR_INPUT
	idate : DATE;
END_VAR
VAR
END_VAR

(*
version 1.2	23 dec 2007
programmer 	hugo
tested by		tobias

calculates the weekday of a week according to ISO8601   
monday = 1 ..... sunday = 7  

*)
IF step7 THEN
	weekday := DWORD_TO_INT((DATE_TO_DWORD(idate)/86400+6) MOD 7) + 1;
ELSE
	weekday := DWORD_TO_INT((DATE_TO_DWORD(idate)/86400+3) MOD 7) + 1;
END_IF;
(* revision history
hm 21.8.06 rev 1.1
	corrected a miscalculation

hm	23.12.2007	rev 1.2
	correction for step7

*)
END_FUNCTION

(* POU Time&Date/period, ST *)
FUNCTION period : BOOL
VAR_INPUT
	d1 : DATE;
	dx : DATE;
	d2 : DATE;
END_VAR
VAR
	day1, day2, dayx : INT;
END_VAR

(*
version 1.3	22. mar. 2008
programmer 	hugo
tested by		tobias

PERIOD checks if a given date is between two dates (d1 and d2) d1 is the starting date and d2 the last date for the period.
the years of the dates are ignored, so the function period cheks for a time period within a year independet of the year.

*)
day1 := day_of_year(d1);
day2 := day_of_year(d2);
dayx := day_of_year(dx);
IF NOT leap_of_Date(dx) AND dayx > 58 THEN dayx := dayx + 1; END_IF;
IF NOT leap_of_Date(d1) AND day1 > 58 THEN day1 :=day1 + 1; END_IF;
IF NOT leap_of_Date(d2) AND day2 > 58 THEN day2 := day2 + 1; END_IF;

IF day2 < day1 THEN
	(* the period spans over the new year *)
	period := dayx <= day2 OR dayx >= day1;
ELSE
	period := dayx >= day1 AND dayx <= day2;
END_IF;

(* code before rev 1.2
yx := year(dx);
p1 := date_add(d1,0,0,0,yx - year(d1));
p2 := date_add(d2,0,0,0,yx - year(d2));

IF p2 >= p1 THEN
	period := dx <= p2  AND dx >= p1;
ELSE
	period := dx <= p2 OR dx >= p1;
END_IF;
*)


(* revision history

hm		19. sep 2007	rev 1.0
	original version

hm		20. sep 2007	rev 1.1
	corrected a problem with leap year

hm		4. jan 2008		rev 1.2
	changed code for better performance

hm		22. mar. 2008	rev 1.3
	function would deliver wrong results when d1, d2 or dx are a leap_year

*)
END_FUNCTION

(* POU XTEST/Testprojekt/TEST Routines/work_week_test, ST *)
FUNCTION work_week_test : BOOL
VAR_INPUT
END_VAR
VAR
	dx: DATE;
	y : ARRAY[0..30] OF INT := 1990,1991,1992,1993,1993,1994,1994,1995,1995,1996,1997,1998,1999,1999,2000,2000,2001,2002,2003,2004,2005,2005,2006,2006,2007,2008,2009,2010,2010,2011,2011;
	w : ARRAY[0..30] OF INT := 1,	1,	 1,   53,  1,   52,	 1,   52,  1,   1,   1,   1,   53,  1,   52,  1,   1,   1,   1,   1,   53,  1,   52,  1,   1,	1,   1,	  53,  1,   52,  1;
	d : ARRAY[0..30] OF INT := 7,	6,	 5,	  3,   10,  2,   9,   1,   8,   7,   5,   4,   3,   10,  2,   9,   7,   6,   5,   4,   2,   9,   1,   8,   7,	6,	 4,	  3,   10,  2,   9;
	i: INT;
	comp: INT;
	d1: DATE;
	day: INT;
	week: INT;
	yr: INT;
END_VAR
work_week_test := TRUE;
FOR i := 0 TO 30 DO
	day := d[i];
	week := w[i];
	yr := y[i];
	d1 := set_Date(yr,1,day);
	comp := work_week(d1);
	IF comp <> week THEN
		work_week_test := FALSE;
		dx := d1;
	END_IF;
	d1 := date_add(d1,-6,0,0,0);
	comp := work_week(d1);
	IF comp <> week THEN
		work_week_test := FALSE;
		dx := d1;
	END_IF;
END_FOR;


(* revision history
hm		26. mar. 2008		rev 1.0
	original release

*)
END_FUNCTION

(* POU Time&Date/work_week, ST *)
FUNCTION work_week : INT
VAR_INPUT
	idate : DATE;
END_VAR
VAR
	d1 : DATE;
	w1 : INT;
	ds: DWORD;
	yr: INT;
	w31: INT;
	w01: INT;
	wm: INT;
END_VAR

(*
version 1.3	16 mar 2008
programmer 	hugo
tested by		tobias

calculates the work week for a given date according to iso8601

*)
(* berechne den 1.1 des jahres von idate. *)
yr := year(idate);
d1 := year_begin(yr);
(* wochentag von d1 *)
w1 := weekday(d1);
(* offset des montags der eletzten KW des vorjahres *)
(* wenn der erste tag des jahres größer als donnerstag ist dann beginnt die letzte kw am montag davor *)
(* wenn der erste tag des jahres ein donnerstag oder kleiner ist beginnt die erste kw 2 montage davor *)
IF w1 < 5 THEN
	ds := DATE_TO_DWORD(d1) - INT_TO_DWORD(w1+6) * 86400;
ELSE
	ds := DATE_TO_DWORD(d1) - INT_TO_DWORD(w1-1) * 86400;
END_IF;

(* kalenderwoche des eingangsdatums *)
work_week := DWORD_TO_INT((DATE_TO_DWORD(idate) - ds) / 604800);

(* korrektur wenn work_week = 0 *)
IF work_week = 0 THEN
	(* work_week needs to be 53 when 1.jan of the year before is thursday or dec 31. is thursday. *)
	(* first and last weekday of a year is equal and one more day for a leap_year. *)
	IF w1 > 1 THEN w31 := w1 - 1; ELSE W31 := 7; END_IF;
	IF leap_year(yr - 1) THEN IF w31 > 1 THEN w01 := W31 - 1; ELSE w1 := 7; END_IF; END_IF;
	(* if first or last day of a year is a thursday, the year has 53 weeks *)
	IF w31 = 4 OR w01 = 4 THEN work_week := 53; ELSE work_week := 52; END_IF;
ELSE
	(* end of year calculation *)
	(* calculated the first and last weekday *)
	IF leap_year(yr) THEN
		IF w1 < 7 THEN w31 := w1 + 1; ELSE w31 := 1; END_IF;
	ELSE
		w31 := w1;
	END_IF;
	(* if first or last day is thursday then the year has 53 weeks otherwise only 52 *)
	IF w31 = 4 OR w1 = 4 THEN wm := 53; ELSE wm := 52; END_IF;
	IF work_week > wm THEN work_week := 1; END_IF;
END_IF;



(* old code before rev 1.2
w1 := weekday(set_Date(year(idate), 1,1));
IF w1 < 5 THEN
	work_week := (day_of_year(idate) + w1 + 5)/7;
ELSE
	work_week := (day_of_year(idate) + w1 - 2)/7;
END_IF
*)


(* revision history

hm 17.1.2007		rev 1.1
	deleted unused variable yday

hm	19. dec 2007	rev 1.2
	changed code for better performance
	changed code to comply with ISO8601

hm	16. mar 2008	rev 1.3
	added type conversions to avoid warnings under codesys 3.0
*)
END_FUNCTION

(* POU XTEST/Testprojekt/math_test, ST *)
FUNCTION_BLOCK math_test
VAR_INPUT
END_VAR
VAR_OUTPUT
	good : BOOL;

END_VAR
VAR CONSTANT
	N : INT := 6;	(* internal resolution in digits *)
END_VAR
VAR
	test: STRING;
	x : REAL;
	y : REAL;
	c : REAL;
	init : BOOL;
	rx : REAL;
END_VAR
IF NOT init THEN
	init := TRUE;
ELSIF NOT good THEN
	RETURN;
ELSE
	good := FALSE;
END_IF;

(* prepare random numbers *)
rx := RDM(rx);

(* test D_trunc *)
test := 'd_trunc';
IF D_TRUNC(0) <> 0 THEN RETURN; END_IF;
IF D_TRUNC(5) <> 5 THEN RETURN; END_IF;
IF D_TRUNC(0.0001) <> 0 THEN RETURN; END_IF;
IF D_TRUNC(0.5) <> 0 THEN RETURN; END_IF;
IF D_TRUNC(0.999) <> 0 THEN RETURN; END_IF;
IF D_TRUNC(-1.5) <> -1 THEN RETURN; END_IF;
IF D_TRUNC(-1.999) <> -1 THEN RETURN; END_IF;
IF D_TRUNC(-1.0001) <> -1 THEN RETURN; END_IF;
IF D_TRUNC(-5) <> -5 THEN RETURN; END_IF;

(* test cmp *)
test := 'cmp';
IF CMP(3.140,3.149,3) = FALSE THEN RETURN; END_IF;
IF CMP(4.2,4.0,2) = TRUE THEN RETURN; END_IF;
IF CMP(0.03140,0.03149,3) = FALSE THEN RETURN; END_IF;
IF CMP(0,0,1) = FALSE THEN RETURN; END_IF;
IF CMP(0.030,0.032,2) = TRUE THEN RETURN; END_IF;

(* check rdm number for range *)
test := 'rdm range';
x := rx;
IF rx < 0 OR rx >= 1 THEN RETURN; END_IF;

(* test acosh 1 <= X < +inv *)
test := 'acosh';
x := rx * 100 + 1;
y := ACOSH(x);
c := LN(SQRT(X*X - 1)+x);
IF NOT CMP(c,y,n) THEN RETURN; END_IF;
test := 'acosh(1)';
y := ACOSH(1);
C := 0;
IF NOT CMP(c,y,n) THEN RETURN; END_IF;

(* test asinh -inv < X < +inv *)
test := 'asinh';
x := (rx-0.5) * 100;
y := asinH(x);
c := LN(SQRT(X*X + 1)+x);
IF NOT CMP(c,y,n) THEN RETURN; END_IF;
test := 'asinh(0)';
y := ASINH(0);
C := 0;
IF NOT CMP(c,y,n) THEN RETURN; END_IF;

(* test atanh -1 < X < +1 *)
test := 'atanh';
x := (rx - 0.5) * 2;
IF x = -1 THEN x := -0.4; END_IF;
y := ATANH(x);
c := LN((1+x)/(1-x))/2;
IF NOT CMP(c,y,n) THEN RETURN; END_IF;
test := 'atanh(0)';
y := ATANH(0);
C := 0;
IF NOT CMP(c,y,n) THEN RETURN; END_IF;

(* test acoth -inv < X < -1 or 1 < X < +inv *)
test := 'acoth X < -1';
x := (rx * 100 - 101);
y := acotH(x);
c := LN((x+1)/(x-1))/2;
IF NOT CMP(c,y,n) THEN RETURN; END_IF;
test := 'acoth X > +1';
x := (rx * -100 + 101);
y := acotH(x);
c := LN((x+1)/(x-1))/2;
IF NOT CMP(c,y,n) THEN RETURN; END_IF;

(* test sinh *)
test := 'sinh';
x := (rx - 0.5) * 5;
y := SINH(x);
c := (EXP(x) - EXP(-x))/2;
IF NOT CMP(c,y,n) THEN RETURN; END_IF;
test := 'sinh(0)';
y := SINH(0);
C := 0;
IF NOT CMP(c,y,n) THEN RETURN; END_IF;

(* test cosh *)
test := 'cosh';
x := (rx - 0.5) * 5;
y := cosH(x);
c := (EXP(x) + EXP(-x))/2;
IF NOT CMP(c,y,n) THEN RETURN; END_IF;
test := 'cosh(0)';
y := COSH(0)-1;
C := 0;
IF NOT CMP(c,y,n) THEN RETURN; END_IF;

(* test tanh *)
test := 'tanh';
x := (rx - 0.5) * 50;
y := tanH(x);
c := 1 - 2 / (EXP(2 * X) + 1);
IF NOT CMP(c,y,n) THEN RETURN; END_IF;
test := 'tanh(0)';
y := tanH(0);
C := 0;
IF NOT CMP(c,y,n) THEN RETURN; END_IF;

(* test coth *)
test := 'coth';
x := (rx - 0.5) * 50;
IF X = 0 THEN X := 1; END_IF;
y := COTH(x);
c := 1 + 2 / (EXP(2 * X) - 1);
IF NOT CMP(c,y,n) THEN RETURN; END_IF;

(* test ceil *)
test := 'ceil';
x := (rx -0.5) * 100;
y := CEIL(x);
c := D_TRUNC(x);
IF x >= 0 THEN c := c + 1; END_IF;
IF NOT CMP(c,y,n) THEN RETURN; END_IF;

(* test ceil2 *)
test := 'ceil2';
x := (rx -0.5) * 100;
y := CEIL2(x);
c := D_TRUNC(x);
IF x >= 0 THEN c := c + 1; END_IF;
IF NOT CMP(c,y,n) THEN RETURN; END_IF;


(* test floor *)
test := 'floor';
x := (rx -0.5) * 100;
y := FLOOR(x);
c := D_TRUNC(x);
IF x < 0 THEN c := c - 1; END_IF;
IF NOT CMP(c,y,n) THEN RETURN; END_IF;

(* test floor *)
test := 'floor2';
x := (rx -0.5) * 100;
y := FLOOR2(x);
c := D_TRUNC(x);
IF x < 0 THEN c := c - 1; END_IF;
IF NOT CMP(c,y,n) THEN RETURN; END_IF;

(* test deg *)
test := 'deg';
x := rx * 2 * 3.14159265358979;
y := DEG(x);
C := X * 180 / 3.14159265358979;
IF NOT CMP(c,y,n) THEN RETURN; END_IF;

(* test rad *)
test := 'rad';
x := rx* 360;
y := Rad(x);
C := X * 3.14159265358979 / 180;
IF NOT CMP(c,y,n) THEN RETURN; END_IF;

(* test differ *)
test := 'differ';
IF differ(10,11,1) = TRUE THEN RETURN; END_IF;
IF differ(11,10,1) = TRUE THEN RETURN; END_IF;
IF differ(10,11,0.999) = FALSE THEN RETURN; END_IF;
IF differ(11,10,0.999) = FALSE THEN RETURN; END_IF;

(* test even *)
test := 'even';
IF even(3) = TRUE THEN RETURN; END_IF;
IF even(-5) = TRUE THEN RETURN; END_IF;
IF even(0) = FALSE THEN RETURN; END_IF;
IF even(10) = FALSE THEN RETURN; END_IF;
IF even(-2) = FALSE THEN RETURN; END_IF;

(* exp10 *)
test := 'exp10';
x := (rx - 0.5) * 4;
y := EXP10(x);
c := EXPT(10,x);
IF NOT CMP(c,y,n) THEN RETURN; END_IF;
test := 'EXP10(10)';
y := EXP10(10);
c := EXPT(10,10);
IF NOT CMP(c,y,n) THEN RETURN; END_IF;

(* test expn *)
test := 'expn^0';
x := (rx -0.5) * 10;
y := EXPN(x,0);
c := EXPT(x,0);
IF NOT CMP(c,y,n) THEN RETURN; END_IF;

test := 'expn^-3';
y := EXPN(x,-3);
c := EXPT(x,-3);
IF NOT CMP(c,y,n) THEN RETURN; END_IF;
test := 'expn^4';
y := EXPN(x,4);
c := EXPT(x,4);
IF NOT CMP(c,y,n) THEN RETURN; END_IF;

(* test fact *)
test := 'fact';
IF FACT(0) <> 1 THEN RETURN; END_IF;
IF FACT(1) <> 1 THEN RETURN; END_IF;
IF FACT(2) <> 2 THEN RETURN; END_IF;
IF FACT(3) <> 6 THEN RETURN; END_IF;
IF FACT(4) <> 24 THEN RETURN; END_IF;
IF FACT(5) <> 120 THEN RETURN; END_IF;
IF FACT(6) <> 720 THEN RETURN; END_IF;
IF FACT(7) <> 5040 THEN RETURN; END_IF;
IF FACT(12) <> 479001600 THEN RETURN; END_IF;

(* test FIB *)
test := 'fib';
IF FIB(0) <> 0 THEN RETURN; END_IF;
IF FIB(1) <> 1 THEN RETURN; END_IF;
IF FIB(2) <> 1 THEN RETURN; END_IF;
IF FIB(3) <> 2 THEN RETURN; END_IF;
IF FIB(4) <> 3 THEN RETURN; END_IF;
IF FIB(10) <> 55 THEN RETURN; END_IF;
IF FIB(20) <> 6765 THEN RETURN; END_IF;
IF FIB(30) <> 832040 THEN RETURN; END_IF;

(* test fract *)
test := 'fract';
x := 3.1415;
y := FRACT(x);
c := 0.1415;
IF NOT CMP(c,y,n) THEN RETURN; END_IF;

(* test gamma *)
test := 'gamma';
x := 2;
y := GAMMA(x);
c := 2;
IF ABS(c-y) > 0.1 THEN RETURN; END_IF;
X := 3;
y := GAMMA(x);
c := 6;
IF ABS(c-y) > 0.2 THEN RETURN; END_IF;
X := 4;
y := GAMMA(x);
c := 24;
IF ABS(c-y) > 0.5 THEN RETURN; END_IF;
X := 10;
y := GAMMA(x);
c := 3628800;
IF ABS(c-y) > 35000 THEN RETURN; END_IF;

(* test hypot *)
test := 'hypot';
x := rx * 100;
y := HYPOT(X,23);
c := SQRT(X*X + 529);
IF NOT CMP(c,y,n) THEN RETURN; END_IF;

(* test inc *)
test := 'inc';
IF INC(3,2,5) <> 5 THEN RETURN; END_IF;
IF INC(3,3,5) <> 0 THEN RETURN; END_IF;
IF INC(3,-3,5) <> 0 THEN RETURN; END_IF;
IF INC(3,-4,5) <> 5 THEN RETURN; END_IF;

(* test langevin *)
test := 'langevin';
Y := LANGEVIN(0);
C := 0;
IF ABS(c-y) > 0.0001 THEN RETURN; END_IF;
Y := LANGEVIN(-5);
C := -0.8;
IF ABS(c-y) > 0.0001 THEN RETURN; END_IF;
Y := LANGEVIN(5);
C := 0.8;
IF ABS(c-y) > 0.0001 THEN RETURN; END_IF;

(* test max3 *)
test := 'max3';
Y := MAX3(1,2,3);
C := 3;
IF NOT CMP(c,y,n) THEN RETURN; END_IF;
Y := MAX3(-1,0,-2);
C := 0;
IF NOT CMP(c,y,n) THEN RETURN; END_IF;
Y := MAX3(3,1,-2);
C := 3;
IF NOT CMP(c,y,n) THEN RETURN; END_IF;
Y := MAX3(1,3,0);
C := 3;
IF NOT CMP(c,y,n) THEN RETURN; END_IF;

(* test min3 *)
test := 'min3';
Y := MIN3(1,2,3);
C := 1;
IF NOT CMP(c,y,n) THEN RETURN; END_IF;
Y := MIN3(-1,0,-2);
C := -2;
IF NOT CMP(c,y,n) THEN RETURN; END_IF;
Y := MIN3(-3,1,-2);
C := -3;
IF NOT CMP(c,y,n) THEN RETURN; END_IF;
Y := MIN3(11,3,10);
C := 3;
IF NOT CMP(c,y,n) THEN RETURN; END_IF;

(* test mid3 *)
test := 'mid3';
Y := MID3(1,2,3);
C := 2;
IF NOT CMP(c,y,n) THEN RETURN; END_IF;
Y := MID3(-1,0,-2);
C := -1;
IF NOT CMP(c,y,n) THEN RETURN; END_IF;
Y := MID3(3,1,-2);
C := 1;
IF NOT CMP(c,y,n) THEN RETURN; END_IF;
Y := MID3(1,3,0);
C := 1;
IF NOT CMP(c,y,n) THEN RETURN; END_IF;

(* test modr *)
test := 'modr';
x := rx * 10;
y := MODR(X,1);
C := FRACT(x);
IF NOT CMP(c,y,n) THEN RETURN; END_IF;

(* test mul_add *)
test := 'mul_add';
X := rx;
Y := MUL_ADD(X,10,20);
C := X * 10 + 20;
IF NOT CMP(c,y,n) THEN RETURN; END_IF;

(* test neg *)
test := 'neg';
X := 13;
IF NEG(13) <> -13 THEN RETURN; END_IF;
X := 0;
IF NEG(0) <> 0 THEN RETURN; END_IF;
X := -4;
IF NEG(-4) <> 4 THEN RETURN; END_IF;

(* test Round *)
test := 'round';
X := 3.14156789;
Y := ROUND(x,0);
C := 3.0;
IF NOT CMP(c,y,n) THEN RETURN; END_IF;
X := 3.14156789;
Y := ROUND(x,5);
C := 3.14157;
IF NOT CMP(c,y,n) THEN RETURN; END_IF;
X := 3.14156789;
Y := ROUND(x,1);
C := 3.1;
IF NOT CMP(c,y,n) THEN RETURN; END_IF;
X := -3.14156789;
Y := ROUND(x,2);
C := -3.14;
IF NOT CMP(c,y,n) THEN RETURN; END_IF;
X := 0.00014;
Y := ROUND(x,4);
C := 0.0001;
IF NOT CMP(c,y,n) THEN RETURN; END_IF;

(* test SGN *)
test := 'sgn';
IF SGN(33) <> 1 THEN RETURN; END_IF;
IF SGN(0) <> 0 THEN RETURN; END_IF;
IF SGN(-4) <> -1 THEN RETURN; END_IF;

(* test sigmoid *)
test := 'sigmoid';
Y := SIGMOID(0);
C := 0.5;
IF NOT CMP(c,y,n) THEN RETURN; END_IF;
Y := SIGMOID(-2);
C := 0.1192029;
IF NOT CMP(c,y,n) THEN RETURN; END_IF;
Y := SIGMOID(2);
C := 0.8807971;
IF NOT CMP(c,y,n) THEN RETURN; END_IF;

(* test sign_I *)
test := 'sign_i';
IF SIGN_I(2) = TRUE THEN RETURN; END_IF;
IF SIGN_I(0) = TRUE THEN RETURN; END_IF;
IF SIGN_I(-3) = FALSE THEN RETURN; END_IF;

(* test sign_R *)
test := 'sign_r';
IF SIGN_R(2) = TRUE THEN RETURN; END_IF;
IF SIGN_R(0) = TRUE THEN RETURN; END_IF;
IF SIGN_R(-3) = FALSE THEN RETURN; END_IF;

(* test sqrtn *)
test := 'sqrtn';
x := rx * 1000;
y := SQRTN(X,5);
c := EXPT(x,0.2);
IF NOT CMP(c,y,n) THEN RETURN; END_IF;

(* test rnd *)
test := 'rnd';
y := RND(-0.00126,2);
C := -0.0013;
IF NOT CMP(c,y,n) THEN RETURN; END_IF;
y := RND(0.00126,2);
C := 0.0013;
IF NOT CMP(c,y,n) THEN RETURN; END_IF;
y := RND(-21.1234567,6);
C := -21.1235;
IF NOT CMP(c,y,n) THEN RETURN; END_IF;
y := RND(0,3);
C := 0;
IF NOT CMP(c,y,n) THEN RETURN; END_IF;
y := RND(21.1234567,6);
C := 21.1235;
IF NOT CMP(c,y,n) THEN RETURN; END_IF;
y := RND(21.1234567,1);
C := 20;
IF NOT CMP(c,y,n) THEN RETURN; END_IF;

(* test window *)
test := 'window';
IF WINDOW(1,2,3) = FALSE THEN RETURN; END_IF;
IF WINDOW(1,1,3) = TRUE THEN RETURN; END_IF;
IF WINDOW(1,3,3) = TRUE THEN RETURN; END_IF;
IF WINDOW(-1,2,3) = FALSE THEN RETURN; END_IF;
IF WINDOW(-5,-2,3) = FALSE THEN RETURN; END_IF;
IF WINDOW(-10,-5,-1) = FALSE THEN RETURN; END_IF;
IF WINDOW(-4,-2,-2) = TRUE THEN RETURN; END_IF;
IF WINDOW(-4,-6,-2) = TRUE THEN RETURN; END_IF;
IF WINDOW(4,8,6) = TRUE THEN RETURN; END_IF;

(* test window2 *)
test := 'window2';
IF WINDOW2(1,2,3) = FALSE THEN RETURN; END_IF;
IF WINDOW2(1,1,3) = FALSE THEN RETURN; END_IF;
IF WINDOW2(1,3,3) = FALSE THEN RETURN; END_IF;
IF WINDOW2(-1,2,3) = FALSE THEN RETURN; END_IF;
IF WINDOW2(-5,-2,3) = FALSE THEN RETURN; END_IF;
IF WINDOW2(-10,-5,-1) = FALSE THEN RETURN; END_IF;
IF WINDOW2(-4,-2,-2) = FALSE THEN RETURN; END_IF;
IF WINDOW2(-4,-5,-2) = TRUE THEN RETURN; END_IF;
IF WINDOW2(-4,-1,-2) = TRUE THEN RETURN; END_IF;
IF WINDOW2(1,0,5) = TRUE THEN RETURN; END_IF;

(* test sinc *)
test := 'sinc';
Y := SINC(0);
C := 1;
IF NOT CMP(c,y,n) THEN RETURN; END_IF;
x := (rx - 0.5)*1000;
Y := SINC(x);
C := SIN(x) / x;
IF NOT CMP(c,y,n) THEN RETURN; END_IF;

(* set output true if there are no errors *)
test := 'finished';
good := TRUE;


(* revision history
hm		26. mar. 2008		rev 1.0
	original release

*)
END_FUNCTION_BLOCK

(* POU Mathematical/ACOSH, ST *)
FUNCTION ACOSH : REAL
VAR_INPUT
	X : REAL;
END_VAR
VAR
END_VAR


(*
version 1.2	16 mar 2008
programmer 	hugo
tested by		tobias

this function calculates the arcus cos hyperbolicus

*)
ACOSH := LN(SQRT(X * X - 1) + X);

(* revision history
hm		12 jan 2007	rev 1.0
	original version

hm		2. dec 2007	rev 1.1
	changed code for better performance

hm		16.3. 2007		rev 1.2
	changed sequence of calculations to improve performance

*)
END_FUNCTION

(* POU Mathematical/ASINH, ST *)
FUNCTION ASINH : REAL
VAR_INPUT
	X : REAL;
END_VAR
VAR
END_VAR


(*
version 1.2	16. mar 2008
programmer 	hugo
tested by		tobias

this function calculates the arcus sin hyperbolicus

*)
ASINH := LN(SQRT(X * X + 1)+X);

(* revision history
hm		12 jan 2007	rev 1.0
	original version

hm		2. dec 2007	rev 1.1
	changed code for better performance

hm		16.3. 2007		rev 1.2
	changed sequence of calculations to improve performance

*)
END_FUNCTION

(* POU Mathematical/ATANH, ST *)
FUNCTION ATANH : REAL
VAR_INPUT
	X : REAL;
END_VAR
VAR
END_VAR


(*
version 1.1	5. jan 2008
programmer 	hugo
tested by		tobias

this function calculates the arcus tangens hyperbolicus

*)
ATANH := LN((1+x)/(1-x)) * 0.5;


(* revision history
hm		12 jan 2007	rev 1.0
	original version

hm		5. jan 2008	rev 1.1
	improved code for better performance
*)
END_FUNCTION

(* POU Mathematical/ACOTH, ST *)
FUNCTION ACOTH : REAL
VAR_INPUT
	X : REAL;
END_VAR
VAR
END_VAR


(*
version 1.1	5. jan 2008
programmer 	hugo
tested by		tobias

this function calculates the arcus cotangens hyperbolicus

*)
acotH := LN((x+1)/(x-1))*0.5;

(* revision history
hm		12 jan 2007	rev 1.0
	original version

hm		5. jan 2008	rev 1.1
	improved code for better performance
*)
END_FUNCTION

(* POU Mathematical/SINH, ST *)
FUNCTION SINH : REAL
VAR_INPUT
	X : REAL;
END_VAR
VAR
END_VAR


(*
version 1.3	11. mar 2008
programmer 	hugo
tested by	tobias

this function calculates the sin hyperbolicus

*)
IF ABS(x) < 2E-3 THEN
	SINH := X;
ELSE
	SINH := (EXP(x) - EXP(-x)) * 0.5;
END_IF;


(* revision history
hm	12.1.2007	rev 1.0
	original version

hm	1.12.2007	rev 1.1
	changed code to improve performance

hm	5. jan 2008	rev 1.2
	further performance improvement

hm	11. mar 2008	rev 1.3
	improved accuracy around 0

*)
END_FUNCTION

(* POU Mathematical/COSH, ST *)
FUNCTION COSH : REAL
VAR_INPUT
	X : REAL;
END_VAR
VAR
	t: REAL;
END_VAR


(*
version 1.2	5. jan 2008
programmer 	hugo
tested by		tobias

this function calculates the cos hyperbolicus

*)
T := EXP(X);
COSH := (1/T + T) * 0.5;

(* revision histroy
hm	12.1.2007	rev 1.0
	original version

hm	1.12.2007	rev 1.1
	changed code to improve performance

hm	5. jan 2008	rev 1.2
	further performance improvement
*)
END_FUNCTION

(* POU Mathematical/TANH, ST *)
FUNCTION TANH : REAL
VAR_INPUT
	X : REAL;
END_VAR
VAR
END_VAR


(*
version 1.2	10. mar 2008
programmer 	hugo
tested by	tobias

this function calculates the tangens hyperbolicus

*)
IF X > 20 THEN
	tanH := 1;
ELSIF X < -20 THEN
	tanH := -1;
ELSE
	tanH := 1 - 2 / (EXP(2 * x) + 1);
END_IF;

(* revision hisdtory
hm		12.1.2007		rev 1.0
	original version

hm		1.12.2007		rev 1.1
	changed code to improve performance

hm		10. mar 2008	rev 1.2
	corrected an error in formula
	extended range of valid inputs to +/- INV
*)
END_FUNCTION

(* POU Mathematical/COTH, ST *)
FUNCTION COTH : REAL
VAR_INPUT
	X : REAL;
END_VAR
VAR
END_VAR


(*
version 1.3	10. mar 2008
programmer 	hugo
tested by		tobias

this function calculates the cotangens hyperbolicus

*)
IF X > 20 THEN
	cotH :=1;
ELSIF X < -20 THEN
	COTH := -1;
ELSE
	COTH := 1 + 2 / (EXP(X * 2) - 1);
END_IF;


(* revision histroy
hm		12.1.2007	rev 1.0
	original version

hm		1.12.2007	rev 1.1
	changed code to improve performance

hm		8. jan 2008	rev 1.2
	further improvement in performance

hm		10. mar 2008	rev 1.3
	extended range of valid inputs to +/- INV
	changed formula for better accuracy
*)
END_FUNCTION

(* POU Mathematical/CEIL, ST *)
FUNCTION CEIL : INT
VAR_INPUT
	X : REAL;
END_VAR
VAR
END_VAR


(*
version 1.0	7 feb 2007
programmer 	hugo
tested by		tobias

This is a rounding function which returns the smallest possible integer which is greater or equal to X.
ceil(3.14) = 4
ceil(-3.14) = -3

*)
CEIL := REAL_TO_INT(x);
IF CEIL < X THEN
        CEIL := CEIL + 1;
END_IF;

(* code before rev 1.1
CEIL := D_TRUNC(X);
IF CEIL < X THEN
	ceil := ceil + 1;
END_IF;
*)

(* revision history
hm		7. feb. 2007	rev 1.0
	original version

hm		21. mar. 2008	rev 1.1
	use REAL_TO_INT instead of trunc for compatibility reasons

*)
END_FUNCTION

(* POU Mathematical/CEIL2, ST *)
FUNCTION CEIL2 : DINT
VAR_INPUT
	X : REAL;
END_VAR
VAR
END_VAR


(*
version 1.0	21. mar. 2008
programmer 	hugo
tested by		tobias

This is a rounding function which returns the smallest possible integer which is greater or equal to X.
ceil2(3.14) = 4
ceil2(-3.14) = -3

*)
CEIL2 := REAL_TO_DINT(x);
IF CEIL2 < X THEN
        CEIL2 := CEIL2 + 1;
END_IF;


(* revision history
hm		21. mar. 2008	rev 1.0
	original version

*)
END_FUNCTION

(* POU Mathematical/FLOOR2, ST *)
FUNCTION FLOOR2 : DINT
VAR_INPUT
	X : REAL;
END_VAR
VAR
END_VAR


(*
version 1.1	21. mar. 2008
programmer 	hugo
tested by		tobias

This is a rounding function which returns the biggest possible integer which is less or equal to X.
floor2(3.14) = 3
floor2(-3.14) = -4

*)
FLOOR2 := REAL_TO_DINT(X);
IF FLOOR2 > X THEN
	FLOOR2 := FLOOR2 - 1;
END_IF;

(* revision history
hm		21. mar. 2008	rev 1.0
	originlal version

*)
END_FUNCTION

(* POU Mathematical/DEG, ST *)
FUNCTION DEG : REAL
VAR_INPUT
	rad : REAL;
END_VAR
VAR
END_VAR
VAR
END_VAR

(*
version 1.1	16 oct 2007
programmer 	hugo
tested by		tobias

this function converts degrees into Radiant
execution time on wago 750 - 841 =  10  us
*)
deg := modR(57.29577951308232 * Rad, 360);

(* revision history
hm	4. aug 2006		rev 1.0
	original version

hm 	16. oct 2007	rev 1.1
	added modr statement which prohibits deg to become bigger than 360

*)
END_FUNCTION

(* POU Mathematical/RAD, ST *)
FUNCTION RAD : REAL
VAR_INPUT
	deg : REAL;
END_VAR
VAR
END_VAR

(*
version 1.0	4 aug 2006
programmer 	hugo
tested by	tobias

this function converts Radiant to degrees

*)
Rad := modR(0.0174532925199433 * deg,PI2);

(* revision history
hm	4. aug 2006
	original version

hm 	16. oct 2007
	added modr statement which prohibits rad to become bigger than 2PI

*)
END_FUNCTION

(* POU Mathematical/MODR, ST *)
FUNCTION MODR : REAL
VAR_INPUT
	in : REAL;
	divi : REAL;
END_VAR

VAR
END_VAR

(*
version 1.2	21. mar. 2008
programmer 	hugo
tested by		tobias

this is a modulo funtion for real numbers
modr(5.5,2.5) = 0.5

*)
IF divi = 0 THEN
	modR := 0;
ELSE
	MODR := in - D_TRUNC(in / divi) * divi;
END_IF;

(* revision history

hm 4.8.2006		rev 1.0

hm 28.1.2007		rev 1.1
	modr(x,0) will deliver the result 0

hm	21. mar 2008	rev 1.2
	use D_trunc for compatibility reasons
*)
END_FUNCTION

(* POU Mathematical/DIFFER, ST *)
FUNCTION DIFFER : BOOL
VAR_INPUT
	in1 : REAL;
	in2 : REAL;
	X : REAL;
END_VAR
VAR
END_VAR

(*
version 1.1	16 mar 2008
programmer 	hugo
tested by		tobias

this function checks if in1 differs more then x from in2
the output is true if abs(in1-in2) > X

*)
DIFFER := ABS(in1 - in2) > X;

(* revision history
hm		8. oct 2006		rev 1.0
	original version

hm		16. mar 2008	rev 1.1
	improverd code for performance

*)
END_FUNCTION

(* POU Mathematical/EXPN, ST *)
FUNCTION EXPN : REAL
VAR_INPUT
	X : REAL;
	N : INT;
END_VAR
VAR
END_VAR

(*
version 1.0	 2 dec 2007
programmer 	hugo
tested by		tobias

this function calculates X to the power of N (Y = X^N) whilke N is an integer
especially on CPU's without a floating point unit this algorythm is about 30 times faster then the IEC standard EXPT() Function

*)
IF n.15 THEN
	(* N is negative *)
	N := ABS(N);
	IF N.0 THEN expn := X; ELSE expn := 1; END_IF;
	N := SHR(N,1);
	WHILE N > 0 DO
		X := X * X;
		IF N.0 THEN expn := expn * X; END_IF;
		N := SHR(N,1);
	END_WHILE;
	expn := 1 / expn;
ELSE;
	IF N.0 THEN expn := X; ELSE expn := 1; END_IF;
	N := SHR(N,1);
	WHILE N > 0 DO
		X := X * X;
		IF N.0 THEN expn := expn * X; END_IF;
		N := SHR(N,1);
	END_WHILE;
END_IF;

(* revision history
hm	4. dec 2007		rev 1.0
	original version

*)
END_FUNCTION

(* POU Mathematical/FACT, ST *)
FUNCTION FACT : DINT
VAR_INPUT
	X : INT;
END_VAR
VAR
	i: INT;
END_VAR

(*
version 1.3	10. mar. 2008
programmer 	hugo
tested by		tobias

this function calculates the factorial of x
this simple factorial only calculates factorials for inputs up to 7
if the input is negative or higher then 7 the output will be -1.

*)
IF x >= 0 AND x < 13 THEN
	FACT := 1;
	i := 2;
	WHILE i <= x DO
		FACT := FACT * i;
		i := i + 1;
	END_WHILE;
ELSE
	FACT := -1;
END_IF;

(* revision history
hm 	4.3.2007			rev 1.1
	changed a critical error where while loop was indefinite.

hm		10.12.2007		rev 1.2
	start value for i has changed to 2 for better performance

hm		10. mar 2008		rev 1.3
	changed output of fact to dint to allow bigger values
*)
END_FUNCTION

(* POU Mathematical/FIB, ST *)
FUNCTION FIB : DINT
VAR_INPUT
	X : INT;
END_VAR
VAR
	t1, t2: DINT;
END_VAR

(*
version 1.3	26. mar. 2008
programmer 	hugo
tested by		tobias

this function calculates the fibonacci sequence

*)
IF X < 0 OR X > 46 THEN
	FIB := -1;
ELSIF x < 2 THEN
	FIB := X;
	RETURN;
ELSE
	(* the fibonacci number is the sum of the two suceeding fibonaci numbers *)
	(* we store the numbers alternatively in t1 and t2 depending on pt *)
	t2 := 1;
	WHILE X > 3 DO
		X := X-2;
		t1 := t1 + t2;
		t2 := t1 + t2;
	END_WHILE;
	IF X > 2 THEN t1 := t1 + t2; END_IF;
	fib := t1 + t2;
END_IF;

(* alternative code for very big numbers

IF X < 31 THEN
	fib := 0.4472136 * (expn(1.618034,X) - expn(-0.618034,X));
ELSE
	fib := 0.4472133 * expn(1.618034,X);
END_IF;

*)

(* revision history
hm		27. dec 2007	rev 1.0
	original version

hm		2. jan 2008	rev 1.1
	deleted unused variable pt

hm		10. mar 2008	rev 1.2
	changed output to dint instead of real

hm		26. mar. 2008	rev 1.3
	function now returns -1 for input < 0 or > 46

*)
END_FUNCTION

(* POU Mathematical/GAMMA, ST *)
FUNCTION GAMMA : REAL
VAR_INPUT
	X : REAL;
END_VAR
VAR
END_VAR

(*
version 1.0	10 dec 2007
programmer 	hugo
tested by		tobias

this function calculates the stirling function which is an approximation for the gamma function

*)
IF X >=0 THEN GAMMA := SQRT(pi2*X)*EXPT(X/E,X); END_IF;

(* revision history
hm	10.12.2007	rev 1.0
	original version

*)
END_FUNCTION

(* POU Mathematical/HYPOT, ST *)
FUNCTION HYPOT : REAL
VAR_INPUT
	X : REAL;
	Y : REAL;
END_VAR
VAR
END_VAR

(*
version 1.0	21 feb 2008
programmer 	hugo
tested by	oscat

this function calculates the pythagorean function

*)
HYPOT := SQRT(x*x + y*y);


(* revision history
hm	21. feb 2008	rev 1.0
	original version

*)
END_FUNCTION

(* POU Mathematical/INC, ST *)
FUNCTION INC : INT
VAR_INPUT
	X : INT;
	D : INT;
	M : INT;
END_VAR
VAR
END_VAR


(*
version 1.1	15. jan 2008
programmer 	hugo
tested by		tobias

This is a increment function which increments the input X by the value D and compares the result with M.
if the output exceeds M it will continue to count from 0 again.

*)
INC := (X + D + M + 1) MOD (M + 1);

(* revision history
hm	7. feb 2007		REV 1.0
	original version

hm	15. jan 2008	rev 1.1
	allow for neagtive increment

*)
END_FUNCTION

(* POU Mathematical/LANGEVIN, ST *)
FUNCTION LANGEVIN : REAL
VAR_INPUT
	X : REAL;
END_VAR
VAR
END_VAR

(*
version 1.1	11 mar 2008
programmer 	hugo
tested by		tobias

this function calculates the langevin function

*)
IF X = 0 THEN
	LANGEVIN := 0;
ELSE
	LANGEVIN := COTH(X) - 1/X;
END_IF;

(* revision history
hm	10.12.2007	rev 1.0
	original version

hm	11. mar 2008	rev 1.1
	changed formula to avoid problems when x = 0
*)
END_FUNCTION

(* POU Mathematical/MAX3, ST *)
FUNCTION MAX3 : REAL
VAR_INPUT
	in1 : REAL;
	in2 : REAL;
	in3 : REAL;
END_VAR
VAR
END_VAR

(*
version 1.0	1 jan 2007
programmer 	hugo
tested by		tobias

this function returns the highest of 3 real values

*)
IF in1 >= in2 AND in1 >= in3 THEN
	max3 := in1;
ELSIF in2 >= in1 AND in2 >= in3 THEN
	max3 := in2;
ELSE
	max3 := in3;
END_IF;
END_FUNCTION

(* POU Mathematical/MIN3, ST *)
FUNCTION MIN3 : REAL
VAR_INPUT
	in1 : REAL;
	in2 : REAL;
	in3 : REAL;
END_VAR
VAR
END_VAR

(*
version 1.0	1 jan 2007
programmer 	hugo
tested by		tobias

this function returns the lowest of 3 real values

*)
IF in1 <= in2 AND in1 <= in3 THEN
	min3 := in1;
ELSIF in2 <= in1 AND in2 <= in3 THEN
	min3 := in2;
ELSE
	min3 := in3;
END_IF;
END_FUNCTION

(* POU Mathematical/MID3, ST *)
FUNCTION MID3 : REAL
VAR_INPUT
	in1 : REAL;
	in2 : REAL;
	in3 : REAL;
END_VAR
VAR
END_VAR

(*
version 1.1	1 jan 2007
programmer 	hugo
tested by		tobias

returns the mid value of 3 real inputs.

*)
IF (in1 <= in2) AND (in1 >= in3) OR (in1 >= in2) AND (in1 <= in3) THEN
	mid3 := in1;
ELSIF (in2 <= in1) AND (in2 >= in3) OR (in2 >= in1) AND (in2 <= in3) THEN
	mid3 := in2;
ELSE
	mid3 := in3;
END_IF;

(*
hm	1.1.2007	rev 1.1
	rewrote the function for better performance

*)
END_FUNCTION

(* POU Mathematical/MUL_ADD, ST *)
FUNCTION MUL_ADD : REAL
VAR_INPUT
	X : REAL;
	K : REAL;
	O : REAL;
END_VAR
VAR
END_VAR

(*
version 1.1	11 nov 2007
programmer 	hugo
tested by		tobias

this function multiplies an input X with K and adds Offset O to the result.

*)
MUL_ADD := X * K + O;

(* revision history
hm	28. feb 2007
	original version

hm	11.nov 2007		rev 1.1
	deleted preset values for K and O this makes no sense for a function

*)
END_FUNCTION

(* POU Mathematical/NEG, ST *)
FUNCTION NEG : INT
VAR_INPUT
	in : INT;
END_VAR
VAR
	X : WORD := 2#1111_1111_1111_1111;
END_VAR

(*
version 1.0	11 nov 2007
programmer 	hugo
tested by		tobias

this function return the value of in multiplied by -1

*)
NEG := WORD_TO_INT(INT_TO_WORD(in - 1) XOR X);

(* revision history
hm 11.11.2007	rev 1.0
	original version

*)
END_FUNCTION

(* POU Mathematical/ROUND, ST *)
FUNCTION ROUND : REAL
VAR_INPUT
	in : REAL;
	N : INT;
END_VAR
VAR
	X: REAL;
END_VAR

(*
version 1.4	16. mar 2008
programmer 	hugo
tested by	tobias

this function rounds a real down to n digits behind the comma.
round(3.1415,1) = 3.1

*)
IF N < 4 THEN
	IF N < 2 THEN
		IF N = 0 THEN X := 1; ELSE X := 10; END_IF;
	ELSE
		IF N = 2 THEN X := 100; ELSE X := 1000; END_IF;
	END_IF;
ELSE
	IF N < 6 THEN
		IF N = 4 THEN X := 10000; ELSE X := 100000; END_IF;
	ELSE
		IF N = 6 THEN X := 1000000; ELSE X := 10000000; END_IF;
	END_IF;
END_IF;

ROUND := DINT_TO_REAL(REAL_TO_DINT(in * X)) / X;


(*
IF in >= 0 THEN
	ROUND := TRUNC(in * X + 0.5) / X;
ELSE
	ROUND := TRUNC(in * X - 0.5) / X;
END_IF;
*)

(* revision history
hm	1. sep 2006	rev 1.0
	original version

hm	2. dec 2007	rev 1.1
	changed code for better performance

hm	8. jan 2008	rev 1.2
	further improvement in performance

hm 11. mar. 2008	rev 1.3
	corrected an error with negative numbers
	use real_to_dint instead of trunc

hm	16. mar 2008	rev 1.4
	added type conversion to avoid warning under codesys 3.0
*)
END_FUNCTION

(* POU Mathematical/SIGMOID, ST *)
FUNCTION SIGMOID : REAL
VAR_INPUT
	X : REAL;
END_VAR
VAR
END_VAR

(*
version 1.1	11.  mar 2008
programmer 	hugo
tested by	tobias

this function calculates the sigmoid function

*)
IF X > 20 THEN
	SIGMOID := 1;
ELSIF x < -85 THEN
	SIGMOID := 0;
ELSE
	SIGMOID := 1 / (1 + EXP(-X));
END_IF;

(* revision history
hm		10.12.2007		rev 1.0
	original version

hm		11. mar. 2008		rev 1.1
	extended range of valid inputs to +inv / -inv

*)
END_FUNCTION

(* POU Mathematical/SIGN_I, ST *)
FUNCTION SIGN_I : BOOL
VAR_INPUT
	in : INT;
END_VAR
VAR
END_VAR

(*
version 1.2	1 dec 2007
programmer 	hugo
tested by	tobias

this function return true if the integer input is negative

*)
sign_I := in.15;

(* revision history
hm 3.3.2007	rev 1.1
	changed method of function for better compatibility to other systems

hm	1.12.2007	rev 1.2
	changed code to improve performance
*)
END_FUNCTION

(* POU Mathematical/SIGN_R, ST *)
FUNCTION SIGN_R : BOOL
VAR_INPUT
	in : REAL;
END_VAR
VAR
	ptr : POINTER TO DWORD;
END_VAR

(*
version 1.2	1 dec 2007
programmer 	hugo
tested by	tobias

this function return true if the real input is negative

*)
ptr := ADR(in);
sign_R := ptr^.31;



(* revision history
hm 19.1.2007	rev 1.1
	changed method of function for better compatibility to other systems

hm	1.12.2007	rev 1.2
	changed code to improve performance
*)
END_FUNCTION

(* POU Mathematical/RND, ST *)
FUNCTION RND : REAL
VAR_INPUT
	X : REAL;
	N : INT;
END_VAR
VAR
	M : REAL;
	LX : INT;
END_VAR

(*
version 1.0	11. mar 2008
programmer 	hugo
tested by	tobias

this function rounds a real down to n digits total.
round(3.1415,2) = 3.1

*)
IF X = 0 THEN
	RND := 0;
ELSE
      LX := CEIL(LOG(ABS(X)));
      M := EXPN(10,N-LX);
      RND := DINT_TO_REAL(REAL_TO_DINT(X * M)) / M;
END_IF;



(* revision history
hm	11. mar 2008	rev 1.0
	original version

*)
END_FUNCTION

(* POU Mathematical/WINDOW, ST *)
FUNCTION WINDOW : BOOL
VAR_INPUT
	low : REAL;
	in : REAL;
	high : REAL;
END_VAR
VAR
END_VAR

(*
	version 1.1	22 jan 2007
	programmer 	hugo
	tested BY	tobias

this checks a signal if the signal is between the upper and lower limit
*)
window := in < high AND in > low;


(* revision history
hm	22.1.2007	rev 1.1
	changed the order of inputs to low, in, high

*)
END_FUNCTION

(* POU Mathematical/WINDOW2, ST *)
FUNCTION WINDOW2 : BOOL
VAR_INPUT
	low : REAL;
	in : REAL;
	high : REAL;
END_VAR
VAR
END_VAR

(*
	version 1.0	31 oct 2007
	programmer 	hugo
	tested BY	tobias

this checks a signal if the signal is between the upper and lower limit including the two limits
*)
WINDOW2 := in <= high AND in >= low;


(* revision history
hm	31.10.2007	rev 1.0
	original version

*)
END_FUNCTION

(* POU Mathematical/SINC, ST *)
FUNCTION SINC : REAL
VAR_INPUT
	X : REAL;
END_VAR
VAR
END_VAR


(*
version 1.0	11. mar 2008
programmer 	hugo
tested by		tobias

this function calculates the sinc function.

*)
IF X = 0 THEN
	SINC := 1;
ELSE
	SINC := SIN(x) / x;
END_IF;


(* revision histroy
hm	11. mar. 2008
	original version

hm	1.12.2007	rev 1.1
	changed code to improove performance

*)
END_FUNCTION

(* POU XTEST/Testprojekt/Measurement_Test, ST *)
FUNCTION_BLOCK Measurement_Test
VAR_INPUT
END_VAR
VAR_OUTPUT
	good: BOOL;
END_VAR
VAR
	test : STRING;
	init: BOOL;
	c: INT;
	start: DWORD;
	timer: DWORD;
	meter1 : meter_test;
END_VAR
IF NOT init THEN
	init := TRUE;
ELSIF NOT good THEN
	RETURN;
ELSE
	good := FALSE;
END_IF;

timer := TIME_TO_DWORD(TIME());

(* test meter *)
test := 'meter';
meter1();
IF NOT meter1.good THEN RETURN; END_IF;




(* set output true if there are no errors *)
test := 'finished';
good := TRUE;


(* revision history
hm		26. mar. 2008		rev 1.0
	original release

*)
END_FUNCTION_BLOCK

(* POU XTEST/Testprojekt/TEST Routines/meter_test, ST *)
FUNCTION_BLOCK meter_test
VAR_INPUT
	tx: TIME;
END_VAR
VAR_OUTPUT
	good : BOOL;
	busy: BOOL;
END_VAR
VAR
	meter1: Meter;
	start: TIME;
	t1: REAL;
	t2: REAL;
END_VAR
tx := TIME();
IF NOT busy THEN
	busy := TRUE;
	meter1(rst := TRUE);
	meter1.RST := FALSE;
	start := Tx;
END_IF;
meter1(m1:=1E9, m2:=4E9, i1:=TRUE, i2:=TRUE, D:= 2, rst:=FALSE);
IF Tx - start >= t#200s THEN
	busy := FALSE;
	t1 := meter1.MX;
	t2 := 2.5E6*TIME_TO_DWORD(tx-start);
	IF NOT CMP(t1, t2, 5) THEN
		good := FALSE;
		RETURN;
	END_IF;
END_IF;

good := TRUE;

(* revision history
hm		26. mar. 2008		rev 1.0
	original release

*)
END_FUNCTION_BLOCK

(* POU Engineering/measurements/Meter, ST *)
FUNCTION_BLOCK Meter
VAR_INPUT
	M1, M2 : REAL;
	I1, I2 : BOOL;
	D : REAL := 1;
	RST : BOOL;
END_VAR
VAR_OUTPUT
	MX : REAL;
END_VAR
VAR RETAIN
	MR : REAL2;
END_VAR
VAR
	MX1, MX2 : REAL; (* current consumption value on M1 and M2 *)
	cycle : TC_S; (* measures the last cycle time in seconds *)
END_VAR

(*
	version 1.2	24. mar. 2008
	programmer 	oscat
	tested BY		oscat

METER measures usage of power or similar values the output MX is the summ of the inputs over time.
MX := sum over time of (I1 * P1 + I2 * P2)/D.
a simple example is the consumption counter for a 2 stage oil burner where stage 1 is 10KW and stage 2 is 20KW.
I1 and I2 decide which value is accounted for, I1 = True only counts P1, I2 is True counts P2 
and I1 and I2 is true counts P1 and P2.
the meter can be used for all kind of consumption meters. P1 and P2 can change on the fly.

*)
(* measure the last cycle time *)
cycle();
(* reset or first time init *)
IF rst THEN
	mr.R1 := 0;
	mr.RX := 0;
ELSE
	(* current consumption measurement *)
	IF I1 THEN MX1 := M1; ELSE MX1 := 0; END_IF;
	IF I2 THEN MX2 := M2; ELSE MX2 := 0; END_IF;
	(* add up the current values in a double real *)
	MR := R2_ADD(MR,(mx1+mx2)/D*cycle.TC);
	(* set the current output value *)
	MX := mr.RX;
END_IF;



(* meter would have a problem when int1 or int2 reach big values
and a short time tick would add a value smaller then the 7 digit resolution of real
therefore the variables m1 and m2 are used to store the counted values 
while the integrators are kept at small values to avoid this overrun

this code was used before rev 1.2
int1(in := M1, Run := I1, rst := rst);
int2(in := M2, Run := I2, rst := rst);
MX := (int1.Out + int2.Out) / D;
*)

(* revision history

hm	16. sep.2007		rev 1.0
	original version

hm	7. feb 2008		rev 1.1
	use new version of ft_int to avoid a counting stop at high values
	deleted unnecessary limits

hm	24. mar. 2008		rev 1.2
	use data_type real2 to extend accuracy to 15 digits total
	do not use ft_int which adds unnecessary overhead
*)
END_FUNCTION_BLOCK

(* POU Engineering/measurements/TC_S, ST *)
FUNCTION_BLOCK TC_S
VAR_INPUT
END_VAR
VAR_OUTPUT
	TC : REAL;
END_VAR
VAR
	init: BOOL;
	tx: DWORD;
	last: DWORD;
END_VAR

(*
	version 1.1	16 mar 2008
	programmer 	hugo
	tested by		tobias

TC_S delivers the time it was last called on the output TC in seconds.

*)
(* read system timer *)
tx := T_PLC_US();

IF NOT init THEN
	init := TRUE;
	TC := 0;
ELSE
	tc := DWORD_TO_REAL(tx - last)*1.0E-6;
END_IF;
last := tx;

(* revision history
hm		13. mar. 2008	rev 1.0
	original version

hm		16. mar 2008	rev 1.1
	added type conversion to avoid warnings under codesys 3.0

*)
END_FUNCTION_BLOCK

(* POU Engineering/measurements/T_PLC_US, ST *)
FUNCTION T_PLC_US : DWORD
VAR CONSTANT
	debug : BOOL := FALSE;
	N : INT := 0;
	offset : DWORD := 0;
END_VAR
VAR
	tx : TIME;
	temp : DWORD := 1;
END_VAR

(*
version 1.1	12 nov 2007
programmer 	hugo
tested by		tobias

T_PLC_US reads the internal PLC timer and return the time, it has the advantage to be able to set a debug mode 
and speed up the counter to test the plc timer overrun which occurs every 50 days respectively 25 days at siemens S7
this routine also allows to correct the behavior of s7 where the internal plc counter will not count all 32 bits.

*)
tx := TIME();
T_PLC_US := TIME_TO_DWORD(Tx)*1000;
(* hier muss die korrektur für step7 stattfinden
plctime muss den vollen wertebereich von time ausnutzen:
wenn bei step7 time -24tage bis plus 24 tage ist dann muss der timer auch beim überlauf auf -24tage springen 
und auf keinen fall auf 0 !!!!
für siemens muss ein weiterer fb im main eingebunden werden der sicherstellt das alle 32 bits durchgezählt werden.
es kann nur ein fb sein den er muss sich das oberste (32te) bit merken.
oder etwa spring s7 bei überlauf auf -24 tage????? dann wäre keine korrektur nötig.
*)
IF debug THEN
	T_PLC_US := (SHL(T_PLC_US,N) OR SHL(temp,N)-1) + Offset;
END_IF;

(* revision history
hm	14.9.2007	rev 1.0
	original version

hm	12. nov 2007	rev 1.1
	added temporaray variable tx because some compilers could not handle time() as an argument

*)
END_FUNCTION

(* POU Mathematical/Double Precision/R2_ADD, ST *)
FUNCTION R2_ADD : REAL2
VAR_INPUT
	X : Real2;
	Y : REAL;
END_VAR
VAR
	temp: REAL;
END_VAR

(*
version 1.0	20. mar. 2008
programmer 	hugo
tested by		tobias

R2_add adds a real to a double real which extends the accuracy of a real to twice as many digits

*)
temp := X.RX;
R2_ADD.RX := Y + X.R1 + X.RX;
R2_ADD.R1 := temp - R2_ADD.RX + Y + X.R1;


(* revision history
hm		20.3.2008	rev 1.0
	original version

*)
END_FUNCTION

(* POU XTEST/Testprojekt/network_test, ST *)
FUNCTION_BLOCK network_test
VAR_INPUT
END_VAR
VAR_OUTPUT
	good : BOOL;
END_VAR
VAR CONSTANT
END_VAR
VAR
END_VAR
good := TRUE;

(* test ip4_decode *)
good := good AND IP4_DECODE('0.0.0.0') = 0;
good := good AND IP4_DECODE('1.2.3.4') = 16#01_02_03_04;
good := good AND IP4_DECODE('255.255.255.255') = 16#FF_FF_FF_FF;
good := good AND IP4_DECODE('256.188.3.4') = 0;
good := good AND IP4_DECODE('1.256.3.4') = 0;
good := good AND IP4_DECODE('1.2.256.4') = 0;
good := good AND IP4_DECODE('1.2.3.256') = 0;
good := good AND IP4_DECODE('1.2.3.4.') = 0;
good := good AND IP4_DECODE('.1.2.3.4.') = 0;
good := good AND IP4_DECODE('1.2.3') = 0;
good := good AND IP4_DECODE('1.A.3.4.') = 0;

(* test is_ip4 *)
good := good AND IS_IP4('0.0.0.0') = FALSE;
good := good AND IS_IP4('192.2.3.0') = TRUE;
good := good AND IS_IP4('255.255.255.255') = TRUE;
good := good AND IS_IP4('256.188.3.4') = FALSE;
good := good AND IS_IP4('1.256.3') = FALSE;
good := good AND IS_IP4('1.A.256.4') = FALSE;
good := good AND IS_IP4('251.188.3.4.1') = FALSE;

(* test ip4_check *)
good := good AND IP4_CHECK(16#01010101,16#01010102,16#FFFFFF00) = TRUE;
good := good AND IP4_CHECK(16#02010101,16#01010102,16#FFFFFF00) = FALSE;
good := good AND IP4_CHECK(16#01020101,16#01010102,16#FF000000) = TRUE;
good := good AND IP4_CHECK(16#02020202,16#01010101,16#000000) = TRUE;


(* revision history
hm		26. mar. 2008		rev 1.0
	original release

*)
END_FUNCTION_BLOCK

(* POU Network/IP4_DECODE, ST *)
FUNCTION IP4_DECODE : DWORD
VAR_INPUT
	str : STRING;
END_VAR
VAR
	d1, d2, d3, d4 : INT;
	s1, s2, s3, s4 : STRING(3);
END_VAR

(*
version 1.0	29. feb 2008
programmer 		kurt
tested by		hugo

IP4_DECODE testet ob ein string eine gültige IPv4 Adresse enthält und gibt die 4 Bytes der IP Adresse als DWORD zurück.

*)
IP4_DECODE := 0;
(* check wheather 3 dots are present *)
IF COUNT_CHAR(str,46) <> 3 THEN RETURN; END_IF;
(* store the positions of the 3 dots *)
d1 := FINDP(str,'.',1);
d2 := FINDP(str,'.',d1+1);
d3 := FINDP(str,'.',d2+1);
IF d1 > 4 OR d2 - d1 > 4 OR d3 - d2 > 4 THEN RETURN; END_IF;
(* store the 3 strings between the dots in d1 .. d4 *)
s1 := LEFT(str,d1-1);
s2 := MID(str,d2-d1-1,d1+1);
s3 := MID(str,d3-d2-1,d2+1);
s4 := RIGHT(str,LEN(str)-d3);
(* check if the 3 strings are numbers only *)
IF NOT IS_NUM(s1) OR NOT IS_NUM(s2) OR NOT IS_NUM(s3) OR NOT IS_NUM(s4) THEN RETURN; END_IF;
(* convert the 4 numbers and check range 0..255 *)
d1 := STRING_TO_INT(s1);
d2 := STRING_TO_INT(s2);
d3 := STRING_TO_INT(s3);
d4 := STRING_TO_INT(s4);
(* check range of numbers *)
IF d1 > 255 OR d2 > 255 OR d3 > 255 OR d4 > 255 THEN RETURN; END_IF;
(* convert to output *)
IP4_DECODE := SHL(INT_TO_DWORD(d1),24) OR SHL(INT_TO_DWORD(d2),16) OR SHL(INT_TO_DWORD(d3),8) OR INT_TO_DWORD(d4);



(* revision history
hm		29. feb 2008	rev 1.0
	original version

*)
END_FUNCTION

(* POU Network/IS_IP4, ST *)
FUNCTION IS_IP4 : BOOL
VAR_INPUT
	str : STRING;
END_VAR
VAR
END_VAR

(*
version 1.0	1. mar 2008
programmer 		kurt
tested by		hugo

IS_IP4 testet ob ein string eine gültige IPv4 Adresse enthält.

*)
IS_IP4 := IP4_DECODE(str) > 0;


(* revision history
hm		1. mar 2008	rev 1.0
	original version

*)
END_FUNCTION

(* POU Network/IP4_CHECK, ST *)
FUNCTION IP4_CHECK : BOOL
VAR_INPUT
	NIP : DWORD;
	LIP : DWORD;
	SM : DWORD;
END_VAR
VAR
END_VAR

(*
version 1.0	4. mar 2008
programmer 	hugo
tested by		oscat

IP4_CHECK testet ob eine Network IP und Local_IP im selben Subnet sind.

*)
IP4_CHECK := (NIP AND sm) = (LIP AND SM);


(* revision history
hm		4. mar 2008	rev 1.0
	original version

*)
END_FUNCTION

(* POU XTEST/Testprojekt/TIME_TEST, ST *)
FUNCTION_BLOCK TIME_TEST
VAR_INPUT
END_VAR
VAR_OUTPUT
	good : BOOL;
END_VAR
VAR
	INIT : BOOL;
	rx : DWORD;
	xt : TIME;
	X : DWORD;
	xtod: TOD;
	xtime: TIME;
	h: INT;
	test: STRING;
	m: INT;
	sec: REAL;
	tmp: REAL;
	N: INT := 6;
	rr: REAL;
END_VAR
IF NOT init THEN
	init := TRUE;
ELSIF NOT good THEN
	RETURN;
ELSE
	good := FALSE;
END_IF;

(* prepare random numbers *)
rx := RDMDW(rx);
rr := RDM(rr);

IF rx <= 86400 THEN
	xtod := DWORD_TO_TOD(rx);
ELSE
	xtod := DWORD_TO_TOD(SHR(rx,6));
END_IF;

xtime := DWORD_TO_TIME(rx);

(* test hour & minute & second *)
test := 'hour & minute & second';
FOR h := 0 TO 23 DO
	x := INT_TO_DWORD(h) * 3600000;
	IF hour(DWORD_TO_TOD(x)) <> h THEN RETURN; END_IF;
	IF hour(DWORD_TO_TOD(x + 3599999)) <> h THEN RETURN; END_IF;
	FOR m := 0 TO 59 DO
		x := INT_TO_DWORD(h) * 3600000 + INT_TO_DWORD(m)*60000;
		IF NOT CMP(second(DWORD_TO_TOD(x)),0,N) THEN RETURN; END_IF;
		IF minute(DWORD_TO_TOD(x)) <> m THEN RETURN; END_IF;
		x := INT_TO_DWORD(h) * 3600000 + INT_TO_DWORD(M) * 60000 + 59999;
		IF NOT CMP(second(DWORD_TO_TOD(x)),59.999,N) THEN RETURN; END_IF;
		IF minute(DWORD_TO_TOD(x)) <> m THEN RETURN; END_IF;
	END_FOR;
END_FOR;

(* test set_tod *)
test := 'set_tod';
IF set_Tod(0,0,0) <> DWORD_TO_TOD(0) THEN RETURN; END_IF;
IF set_Tod(1,0,0) <> DWORD_TO_TOD(3600000) THEN RETURN; END_IF;
IF set_Tod(23,59,59.999) <> DWORD_TO_TOD(86399999) THEN RETURN; END_IF;
h := hour(xtod);
m := minute(xtod);
sec := second(xtod);
IF set_Tod(h,m,sec) <> xtod THEN RETURN; END_IF;


(* test minute hour second *)
test := ' minute hour second ';
h := hour(xtod);
m := minute(xtod);
sec := second(xtod);
IF set_Tod(h,m,sec) <> xtod THEN RETURN; END_IF;

(* test hour_to_time *)
test := 'hour_to_time';
tmp := rr * 100;
xt := hour_to_time(tmp);
IF NOT CMP(TIME_TO_REAL(xt), REAL_TO_DINT(tmp * 3600000),N) THEN RETURN; END_IF;

(* test minute_to_time *)
test := 'minute_to_time';
tmp := rr * 100;
xt := minute_to_time(tmp);
IF NOT CMP(TIME_TO_REAL(xt),REAL_TO_DINT(tmp * 60000),N) THEN RETURN; END_IF;

(* test second_to_time *)
test := 'second_to_time';
tmp := rr * 100;
xt := second_to_time(tmp);
IF NOT CMP(TIME_TO_REAL(xt), REAL_TO_DINT(tmp * 1000),N) THEN RETURN; END_IF;

(* test day_to_time *)
test := 'day_to_time';
tmp := rr*10;
xt := day_to_time(tmp);
IF NOT CMP(TIME_TO_REAL(xt), REAL_TO_DINT(tmp * 86400000),N) THEN RETURN; END_IF;

(* test hour_to_tod *)
test := 'hour_to_tod';
tmp := rr * 100;
xtod := hour_to_tod(tmp);
IF NOT CMP(TOD_TO_REAL(xtod),REAL_TO_DINT(tmp * 3600000),N) THEN RETURN; END_IF;

(* test multime *)
test := 'multime';
xt := multime(DWORD_TO_TIME(rx), rr);
IF TIME_TO_DWORD(xt) <> REAL_TO_DWORD(DWORD_TO_REAL(rx) * rr) THEN RETURN; END_IF;



(* set output true if there are no errors *)
test := 'finished';
good := TRUE;


(* revision history
hm		26. mar. 2008		rev 1.0
	original release

*)
END_FUNCTION_BLOCK

(* POU Time&Date/set_Tod, ST *)
FUNCTION set_Tod : TOD
VAR_INPUT
	hour : INT;
	minute : INT;
	second : REAL;
END_VAR
VAR
END_VAR

(*
version 1.5	16. mar 2008
programmer 	hugo
tested by		tobias

creates tod from hour minute and second 

*)
set_Tod := DWORD_TO_TOD(REAL_TO_DWORD(second * 1000) + INT_TO_DWORD(minute) * 60000 + INT_TO_DWORD(hour) * 3600000);

(* revision history

hm		4.aug.2006		rev 1.0
	original version

hm		11. sep 2007	rev 1.1
	changed coding to avoid a compiler warning under twincat.

hm		1. nov 2007	rev 1.2
	changed coding to avoid possible overrun situation on möller ecp4

hm		2. Nov	2007	rev 1.3
	changed dword to DINT in calcualtion to avoid warnings with some compilers

hm		14. mar 2008	rev 1.4
	changed code to avoid rounding problem at last digit of millisecond

hm		16. mar. 2008	rev 1.5
	added type conversions to avoid warning under codesys 3.0
*)
END_FUNCTION

(* POU Time&Date/hour_to_time, ST *)
FUNCTION hour_to_time : TIME
VAR_INPUT
	input : REAL;
END_VAR
VAR
END_VAR

(*
version 1.1	14 mar 2008
programmer 	hugo
tested by		tobias

converts an amount of hours in real to time

*)
hour_to_time := DWORD_TO_TIME(REAL_TO_DWORD(input * 3600000));


(* revision history
hm		4. aug 2006	rev 1.0
	original version

hm		14. mar 2008	rev 1.1
	rounded the input after the last digit

*)
END_FUNCTION

(* POU Time&Date/minute_to_time, ST *)
FUNCTION minute_to_time : TIME
VAR_INPUT
	input : REAL;
END_VAR
VAR
END_VAR

(*
version 1.1	14 mar 2008
programmer 	hugo
tested by		tobias

converts an amount of minutes in real to time
execution time on wago 750-841 =  17us
*) 
minute_to_time := DWORD_TO_TIME(REAL_TO_DWORD(input * 60000));


(* revision history
hm		4. aug 2006	rev 1.0
	original version

hm		14. mar 2008	rev 1.1
	rounded the input after the last digit

*)
END_FUNCTION

(* POU Time&Date/second_to_time, ST *)
FUNCTION second_to_time : TIME
VAR_INPUT
	input : REAL;
END_VAR
VAR
END_VAR

(*
version 1.1	44 mar 2008
programmer 	hugo
tested by		tobias

converts an amount of seconds in real to time
execution TIME on wago 750-841 =  17us 

*)
second_to_time := DWORD_TO_TIME(REAL_TO_DWORD(input * 1000));

(* revision history
hm		4. aug 2006	rev 1.0
	original version

hm		14. mar 2008	rev 1.1
	rounded the input after the last digit
*)
END_FUNCTION

(* POU Time&Date/day_to_time, ST *)
FUNCTION day_to_time : TIME
VAR_INPUT
	input : REAL;
END_VAR
VAR
END_VAR

(*
version 1.0	4 aug 2006
programmer 	hugo
tested by		tobias

converts an amount of days in real to time 
*)
day_to_time := DWORD_TO_TIME(REAL_TO_DWORD(input * 86400000));
END_FUNCTION

(* POU Time&Date/hour_to_tod, ST *)
FUNCTION hour_to_tod : TOD
VAR_INPUT
	input : REAL;
END_VAR
VAR
END_VAR

(*
version 1.1	14 aug 2008
programmer 	hugo
tested by		tobias

converts an amount of hours in real to time of day TOD.

*)
hour_to_tod := DWORD_TO_TOD(REAL_TO_DWORD(input * 3600000));


(* revision history
hm		4. aug 2006	rev 1.0
	original version

hm		14. mar 2008	rev 1.1
	rounded the input after the last digit

*)
END_FUNCTION

(* POU Time&Date/multime, ST *)
FUNCTION multime : TIME
VAR_INPUT
	t : TIME;
	M : REAL;
END_VAR
VAR
END_VAR


(*
version 1.1	14 mar 2008
programmer 	hugo
tested by		tobias

multiplies a time by a real number and returns a time
*)
multime := DWORD_TO_TIME(REAL_TO_DWORD(DWORD_TO_REAL(TIME_TO_DWORD(t))*M));

(* revision history
hm		2. oct 2006	rev 1.0
	original version

hm		14. mar 2008	rev 1.1
	rounded the result after the last digit

*)
END_FUNCTION

(* POU XTEST/Baustein Tests/air_test, CFC *)
PROGRAM air_test
VAR
	temp: REAL := 70;
	den: REAL;
	den1: REAL;
	ent: REAL;
	cp: REAL;
	rh: REAL := 0.5;
	P: REAL := 101325;
	ice: BOOL;
	SDx: REAL;
	enth: REAL;
END_VAR
VAR (* helpers for the ST form of the networks *)
	_t78 : REAL;
	_t90 : REAL;
END_VAR
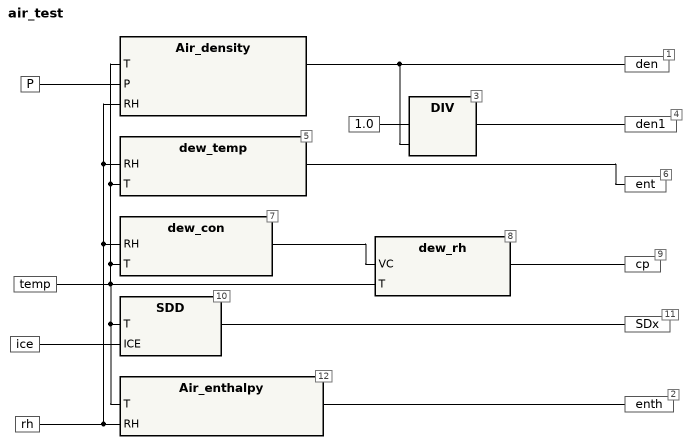
_CFC_ (* Continuous Function Chart, elements in execution order *)
#0 Air_density(T: temp, P: P, RH: rh)
#1 den <= #0
#2 enth <= #12
#3 DIV(1.0, #0)
#4 den1 <= #3
#5 dew_temp(RH: rh, T: temp)
#6 ent <= #5
#7 dew_con(RH: rh, T: temp)
#8 dew_rh(VC: #7, T: temp)
#9 cp <= #8
#10 SDD(T: temp, ICE: ice)
#11 SDx <= #10
#12 Air_enthalpy(T: temp, RH: rh)
_END_CFC_
(* the same logic as Structured Text *)
_t78 := Air_density(T := temp, P := P, RH := rh);
den := _t78;
enth := _t90;
den1 := 1.0 / _t78;
ent := dew_temp(RH := rh, T := temp);
cp := dew_rh(VC := dew_con(RH := rh, T := temp), T := temp);
SDx := SDD(T := temp, ICE := ice);
_t90 := Air_enthalpy(T := temp, RH := rh);
END_PROGRAM

(* POU Building/HLK/Air_density, ST *)
FUNCTION Air_density : REAL
VAR_INPUT
	T : REAL;
	P : REAL;
	RH : REAL;
END_VAR
VAR CONSTANT
	RL : REAL := 287.05;
	RX : REAL := 3.773319E-3;
END_VAR
VAR
END_VAR

(*
version 1.1	4 dec 2007
programmer 	hugo
tested by		tobias

this function calculates the air density between 0 and 100 deg C

*)
Air_density := PN * (1 - RH * SDD(T, TRUE) * RX / P) / (RL * ( T - TK));

(* original code used for rev 1.0

SDD := SDD(T,FALSE);
RF := RL / (1- RH*SDD/P*RX);
Air_density := P / (RF * (T-TK));

*)

(* revision history

hm	29.10.2007		rev 1.0
	original version

hm	4.12.2007		rev 1.1
	changed code for better performance

*)
END_FUNCTION

(* POU Building/HLK/SDD, ST *)
FUNCTION SDD : REAL
VAR_INPUT
	T : REAL;
	ICE: BOOL;
END_VAR
VAR CONSTANT
END_VAR
VAR
END_VAR

(*
version 1.1	2 dec 2007
programmer 	hugo
tested by		tobias

this function calculates the vapor saturation pressure for moist Air over ice or water

*)
IF ice THEN
	SDD := 611.153 * EXP(22.4433 * T / (272.186 + T));
ELSE
	SDD := 611.213 * EXP(17.5043 * T / (241.2 + T));
END_IF;

(* old code used in rev 1.0
IF ice THEN
	SDD := 611.153 * exp10(9.747*T / (272.186 + T));
ELSE
	SDD := 611.213 * exp10(7.602*T / (241.2 + T));
END_IF;
*)


(* revision history

hm 29 oct 2007		rev 1.0
	original version

hm	2. dec 2007		rev 1.1
	changed code for better performance
*)
END_FUNCTION

(* POU Building/HLK/dew_temp, ST *)
FUNCTION dew_temp : REAL
VAR_INPUT
	RH : REAL;
	T : REAL;
END_VAR
VAR CONSTANT
	a : REAL := 7.5;
	b : REAL := 237.3;
END_VAR
VAR
	V : REAL;
END_VAR

(*
version 1.4	8 jan 2008
programmer 	hugo
tested by		tobias

this function calculates the dew point for air given the temperature and relative humidity.
dew_temp(60,0.25) = 16.7 °C.
which means the dew point for air with 25° and 60% RH is at 16.7 °C.


*)
IF rh > 0 THEN
(*	old code was rewritten for better performance
	SDD := 6.1078*EXPT(10,(a*T)/(b+T));
	DD := RH/100 * SDD;
	V := LOG(DD/6.1078);
	dew_temp := b*V/(a-v);
*)
	V := LOG(RH * 0.01 * exp10((a*T)/(b+T)));
	dew_temp := b*V/(a-V);
ELSE
	dew_temp:= -TK;
END_IF;

(* revision history

hm		2.10.2006	rev 1.0
	original version created

hm		29.4.2007	rev 1.1
	checked for rh not to be 0 because log(0) is not defined

hm		13.9.2007	rev 1.2
	code rewritten for better performance

hm		2. dec 2007	rev 1.3
	changed code for better performance

hm		8. jan 2008	rev 1.4
	further improvement in performance
*)

(*
Bezeichnungen:
r = relative Luftfeuchte
T = Temperatur in °C
TK = Temperatur in Kelvin (TK = T + 273.15)
TD = Taupunkttemperatur in °C
DD = Dampfdruck in hPa
SDD = Sättigungsdampfdruck in hPa

Parameter:
a = 7.5, b = 237.3 für T >= 0
a = 7.6, b = 240.7 für T < 0 über Wasser (Taupunkt)
a = 9.5, b = 265.5 für T < 0 über Eis (Frostpunkt)

R* = 8314.3 J/(kmol*K) (universelle Gaskonstante)
mw = 18.016 kg (Molekulargewicht des Wasserdampfes)
AF = absolute Feuchte in g Wasserdampf pro m3 Luft

Formeln:

   1. SDD(T) = 6.1078 * 10^((a*T)/(b+T))
   2. DD(r,T) = r/100 * SDD(T)
   3. r(T,TD) = 100 * SDD(TD) / SDD(T)
   4. TD(r,T) = b*v/(a-v) mit v(r,T) = log10(DD(r,T)/6.1078)
   5. AF(r,TK) = 10^5 * mw/R* * DD(r,T)/TK; AF(TD,TK) = 10^5 * mw/R* * SDD(TD)/TK 

*)
END_FUNCTION

(* POU Building/HLK/dew_con, ST *)
FUNCTION dew_con : REAL
VAR_INPUT
	RH : REAL;
	T : REAL;
END_VAR
VAR CONSTANT
END_VAR
VAR
END_VAR

(*
version 1.2	2 dec 2007
programmer 	hugo
tested by		tobias

this function calculates the water concentratin in air for a given temperature and relative humidity.
the output states the concentration of water vapor in air in Gramms / qubic meter.

*)
IF rh > 0 THEN
(*	this code is good to read but need to be improoved
	SDD := 6.1078*EXPT(10,(a*T)/(b+T));
	DD := RH/100 * SDD;
	V := LOG(DD/6.1078);
	TD := b*V/(a-v);
	dew_con := 0.1 * mw / RU * DD / (T - TK);
*)
	dew_con := 2.166824303E-2 * RH * SDD(T,FALSE)  / (T - TK);
ELSE
	dew_con := 0;
END_IF;

(*
Bezeichnungen:
r = relative Luftfeuchte
T = Temperatur in °C
TK = Temperatur in Kelvin (TK = T + 273.15)
TD = Taupunkttemperatur in °C
DD = Dampfdruck in hPa
SDD = Sättigungsdampfdruck in hPa

Parameter:
a = 7.5, b = 237.3 für T >= 0
a = 7.6, b = 240.7 für T < 0 über Wasser (Taupunkt)
a = 9.5, b = 265.5 für T < 0 über Eis (Frostpunkt)

R* = 8314.3 J/(kmol*K) (universelle Gaskonstante)
mw = 18.016 kg (Molekulargewicht des Wasserdampfes)
AF = absolute Feuchte in g Wasserdampf pro m3 Luft

Formeln:

   1. SDD(T) = 6.1078 * 10^((a*T)/(b+T))
   2. DD(r,T) = r/100 * SDD(T)
   3. r(T,TD) = 100 * SDD(TD) / SDD(T)
   4. TD(r,T) = b*v/(a-v) mit v(r,T) = log10(DD(r,T)/6.1078)
   5. AF(r,TK) = 10^5 * mw/R* * DD(r,T)/TK; AF(TD,TK) = 10^5 * mw/R* * SDD(TD)/TK 

*)

(* revision history

hm 29 apr 2007		rev 1.0
	original version

hm	13.sep 2007		rev 1.1
	improoved coding for speed
	deleted unused variabled SDD,DD,V, TD

hm	2. dec 2007		rev 1.2
	changed code for better performance
	output is now in Gramms / Qubic meter
*)
END_FUNCTION

(* POU Building/HLK/dew_rh, ST *)
FUNCTION dew_rh : REAL
VAR_INPUT
	VC : REAL;
	T : REAL;
END_VAR

(*
version 1.1	2 dec 2007
programmer 	hugo
tested by		tobias

this function calculates the relative humidity in air for a given temperature in °C and vapor concentration in Kg/m³..

*)
dew_rh := LIMIT(0,VC / dew_con(1,T),100);

(* code before rev 1.1
dew_rh := VC / dew_con(100,T) * 100;
IF dew_rh > 100 THEN dew_rh := 100; END_IF;
*)

(* revision history
hm		29. apr 2007	rev 1.0
	original version

hm		2. 12. 2007		rev 1.1
	new code for better performance

*)
END_FUNCTION

(* POU Building/HLK/Air_enthalpy, ST *)
FUNCTION Air_enthalpy : REAL
VAR_INPUT
	T : REAL;
	RH : REAL;
END_VAR
VAR CONSTANT
	CPL : REAL := 1.00482;
	CW : REAL := 1.86;
	LH : REAL := 2500.78;
END_VAR
VAR
END_VAR

(*
version 1.1	2 nov 2007
programmer 	hugo
tested by		tobias

this function calculates the enthalpy for humid air between 0 and 100 deg C

*)
Air_enthalpy := CPL * T + (CW * T + LH) * dew_con(RH,T);

(* revision history

hm	31.10.2007		rev 1.0
	original version

hm	2.11.2007		rev 1.1
	deleted unused variable RF

hm	2.12.2007		rev 1.2
	changed code for better performance
*)
END_FUNCTION

(* POU XTEST/Baustein Tests/bcd_test, CFC *)
PROGRAM bcd_test
VAR
	strbcd: STRING;
	inout: INT;
	inx: INT;
END_VAR
VAR_INPUT

END_VAR
VAR (* helpers for the ST form of the networks *)
	_t28 : BCD;
	_t27 : INT;
END_VAR
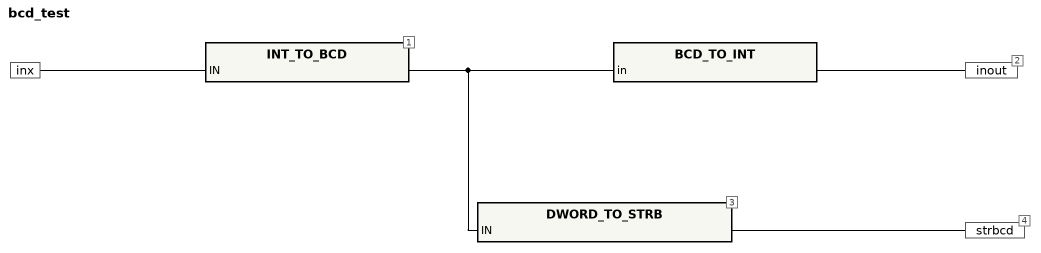
_CFC_ (* Continuous Function Chart, elements in execution order *)
#0 BCD_TO_INT(in: #1)
#1 INT_TO_BCD(IN: inx)
#2 inout <= #0
#3 DWORD_TO_STRB(IN: #1)
#4 strbcd <= #3
_END_CFC_
(* the same logic as Structured Text *)
_t27 := BCD_TO_INT(in := _t28);
_t28 := INT_TO_BCD(IN := inx);
inout := _t27;
strbcd := DWORD_TO_STRB(IN := _t28);
END_PROGRAM

(* POU Logic/gate logic/BCD_TO_INT, ST *)
FUNCTION BCD_TO_INT : INT
VAR_INPUT
	in : BYTE;
END_VAR
VAR
END_VAR

(*
version 1.0	13 dec 2007
programmer 	hugo
tested by		tobias

this function converts a two digit bcd number into an integer.
*)
	BCD_TO_INT := (in AND 16#0F) + (SHR(in,4) * 10);

(* revision history
hm	13.12.2007
	original version

*)
END_FUNCTION

(* POU Logic/gate logic/INT_TO_BCD, ST *)
FUNCTION INT_TO_BCD : BYTE
VAR_INPUT
	IN : INT;
END_VAR
VAR
END_VAR

(*
version 1.0	17 jan 2007
programmer 	hugo
tested by		tobias

this function converts an integer into a two digit bcd number.
*)
INT_TO_BCD := INT_TO_BYTE(SHL(TRUNC(in/10),4) + (in MOD 10));

(* revision history
hm	13.12.2007
	original version

*)
END_FUNCTION

(* POU XTEST/Baustein Tests/blind_test, CFC *)
PROGRAM blind_test
VAR
	up: BOOL;
	dn: BOOL;
	x1: blind_scene;
	mu: BOOL;
	md: BOOL;
	pos: BYTE;
	ang: BYTE;
	x2: blind_security;
	esr: BYTE;
	fire: BOOL;
	wind: BOOL;
	alarm: BOOL;
	rain: BOOL;
	x3: blind_control;
	x5: blind_input;
	p: BYTE;
	a: BYTE;
	IN: BOOL;
	utc: DT;
	X7: blind_night;
	x8: sun_time;
	Door: BOOL;
	x9: sun_pos;
	x10: BLIND_SHADE;
	S_write: BOOL;
	S_enable: BOOL;
	scene: BYTE;
	sun: BOOL;
	ex: BOOL;
END_VAR
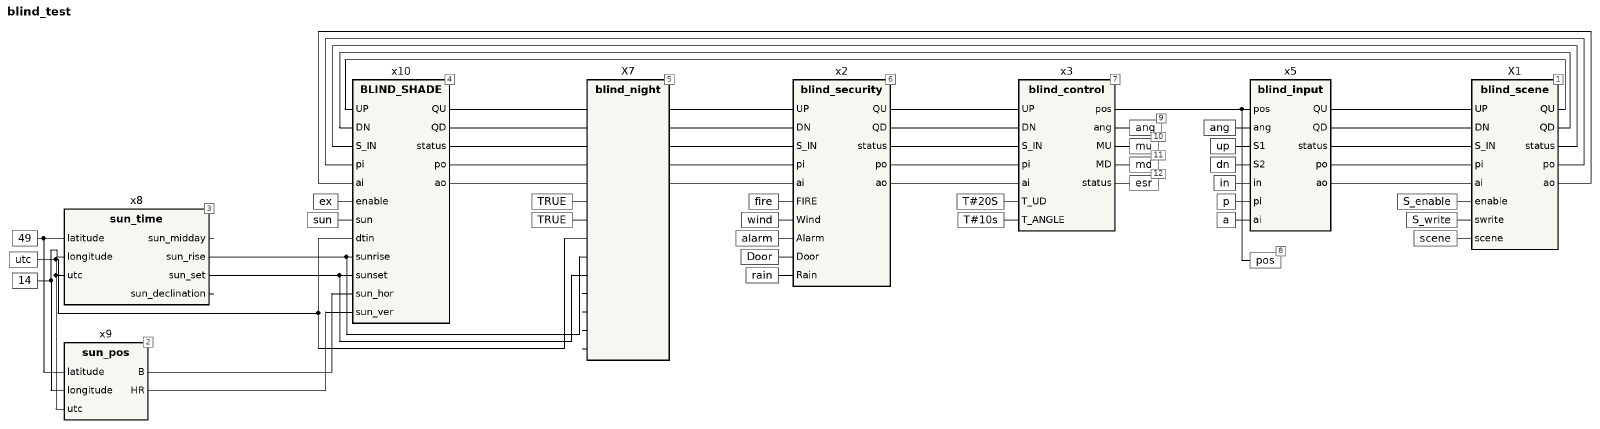
_CFC_ (* Continuous Function Chart, elements in execution order *)
#0 x5:blind_input(pos: #7.pos, ang: ang, S1: up, S2: dn, in: in, pi: p, ai: a, click_mode := TRUE, click_time := T#250ms, manual_timeout := T#10s)
#1 X1:blind_scene(UP: #0.QU, DN: #0.QD, S_IN: #0.status, pi: #0.po, ai: #0.ao, enable: S_enable, swrite: S_write, scene: scene)
#2 x9:sun_pos(latitude: 49, longitude: 14, utc: utc)
#3 x8:sun_time(latitude: 49, longitude: 14, utc: utc)
#4 x10:BLIND_SHADE(UP: #1.QU, DN: #1.QD, S_IN: #1.status, pi: #1.po, ai: #1.ao, enable: ex, sun: sun, dtin: utc, sunrise: #3.sun_rise, sunset: #3.sun_set, sun_hor: #2.B, sun_ver: #2.HR, direction := 180, slat_width := 60, Slat_spacing := 60)
#5 X7:blind_night(#4.QU, #4.QD, #4.status, #4.po, #4.ao, TRUE, TRUE, utc, #3.sun_rise, #3.sun_set, -, -, -, -)
#6 x2:blind_security(UP: #5.out 1, DN: #5.out 2, S_IN: #5.out 3, pi: #5.out 4, ai: #5.out 5, FIRE: fire, Wind: wind, Alarm: alarm, Door: Door, Rain: rain, Alarm_UP := TRUE)
#7 x3:blind_control(UP: #6.QU, DN: #6.QD, S_IN: #6.status, pi: #6.po, ai: #6.ao, T_UD: T#20S, T_ANGLE: T#10s, sens := 5, T_Lockout := T#3s)
#8 pos <= #7.pos
#9 ang <= #7.ang
#10 mu <= #7.MU
#11 md <= #7.MD
#12 esr <= #7.status
_END_CFC_
END_PROGRAM

(* POU Building/Jalousie/blind_scene, ST *)
FUNCTION_BLOCK blind_scene
VAR_INPUT
	UP, DN : BOOL;
	S_IN : BYTE;
	pi, ai : BYTE;
	enable : BOOL;
	swrite : BOOL;
	scene : BYTE;
END_VAR
VAR_INPUT CONSTANT
END_VAR
VAR_OUTPUT
	QU, QD : BOOL;
	status : BYTE;
	po, ao : BYTE;
END_VAR
VAR RETAIN
	sx : ARRAY[0..15,0..2] OF BYTE;
END_VAR
VAR_TEMP
	x : BYTE;

END_VAR

(*
version 1.1	29. jan 2008
programmer 	hugo
tested by		tobias


*)
(* delete all bits except the lower 4 of scene *)
x := scene AND 16#0F;

IF enable AND sx[x,2] > 0 AND UP AND DN THEN
	po := sx[x,0];
	ao := sx[x,1];
	status := 160 + x;  (* Status number is 160 to 175 for the 16 scenes *)
	QU := TRUE;
	QD := TRUE;
ELSE
	QU := UP;
	QD := DN;
	status := S_IN;
	po := pi;
	ao := ai;
END_IF;

(* write scene if necessary *)
IF swrite THEN
	status := 176;		(* write scene *)
	sx[x,0] := pi;
	sx[x,1] := ai;
	IF enable THEN sx[x,2] := 1; ELSE sx[x,2] := 0; END_IF; (* if sx[x,2] = 0 the scene is disabled *)
END_IF;


(* revision history
hm	24. oct 2007	rev 1.0
	original release

hm		29.1.2008	rev 1.1
	replaced shr/shl with and for better performance
*)
END_FUNCTION_BLOCK

(* POU Building/Jalousie/blind_security, ST *)
FUNCTION_BLOCK blind_security
VAR_INPUT
	UP, DN : BOOL;
	S_IN : BYTE;
	pi, ai : BYTE;
	FIRE : BOOL;
	Wind : BOOL;
	Alarm : BOOL;
	Door : BOOL;
	Rain : BOOL;
END_VAR
VAR_INPUT CONSTANT
	Alarm_UP : BOOL := TRUE;
	WIND_UP :BOOL := TRUE;
	RAIN_UP : BOOL := FALSE;
END_VAR
VAR_OUTPUT
	QU, QD : BOOL;
	status : BYTE;
	po, ao : BYTE;
END_VAR
VAR
END_VAR

(*
version 1.2	12. feb 2008
programmer 	hugo
tested by		tobias


*)
IF Fire THEN
	QU := TRUE;
	QD := FALSE;
	status := 111;
ELSIF Wind THEN
	QU := Wind_up;
	QD := NOT wind_up;
	status := 112;
ELSIF alarm THEN
	QU := Alarm_up;
	QD := NOT Alarm_up;
	status := 113;
ELSIF Door THEN
	QU := TRUE;
	QD := FALSE;
	status := 114;
ELSIF Rain AND NOT (up XOR dn) THEN
	QU := rain_up;
	QD := NOT rain_up;
	status := 115;
ELSE
	QU := UP;
	QD := DN;
	status := S_IN;
	po := pi;
	ao := ai;
END_IF;


(* revision history
hm	29. sep 2007	rev 1.0
	original release

hm	6. oct 2007		rev 1.1
	added pos and angle inputs and outputs
	manual will override rain position
	alarm position can now be configured

hm		12. feb. 2008	rev 1.2
	added config variables rain_up and wind_up
	position for rain and wind is now configurable
*)
END_FUNCTION_BLOCK

